LIN {X 0,Y 417.103,Z 397.247,A -85,B 0,C 180,E1 -10165.167,E2 -10165.167} C_VEL
LIN {X 0,Y 417.015,Z 399.098,A -85,B 0,C 180,E1 -10166.135,E2 -10166.135} C_VEL
LIN {X 0,Y 417.032,Z 400.492,A -85,B 0,C 180,E1 -10167.102,E2 -10167.102} C_VEL
LIN {X 0,Y 417.07,Z 401.489,A -85,B 0,C 180,E1 -10168.069,E2 -10168.069} C_VEL
LIN {X 0,Y 417.035,Z 402.093,A -85,B 0,C 180,E1 -10169.035,E2 -10169.035} C_VEL
LIN {X 0,Y 417.032,Z 402.291,A -85,B 0,C 180,E1 -10170,E2 -10170} C_VEL
LIN {X 0,Y 417.071,Z 401.439,A -85,B 0,C 180,E1 -10171.932,E2 -10171.932} C_VEL
LIN {X 0,Y 417.033,Z 400.426,A -85,B 0,C 180,E1 -10172.898,E2 -10172.898} C_VEL
LIN {X 0,Y 417.016,Z 398.993,A -85,B 0,C 180,E1 -10173.866,E2 -10173.866} C_VEL
LIN {X 0,Y 417.09,Z 396.015,A -85,B 0,C 180,E1 -10175.318,E2 -10175.318} C_VEL
LIN {X 0,Y 417.18,Z 391.978,A -85,B 0,C 180,E1 -10176.773,E2 -10176.773} C_VEL
LIN {X 0,Y 417.476,Z 385.766,A -85,B 0,C 180,E1 -10178.471,E2 -10178.471} C_VEL
LIN {X 0,Y 417.86,Z 378.993,A -85,B 0,C 180,E1 -10179.927,E2 -10179.927} C_VEL
LIN {X 0,Y 418.41,Z 370.585,A -85,B 0,C 180,E1 -10181.383,E2 -10181.383} C_VEL
LIN {X 0,Y 419.028,Z 361.919,A -85,B 0,C 180,E1 -10182.594,E2 -10182.594} C_VEL
LIN {X 0,Y 419.708,Z 351.481,A -85,B 0,C 180,E1 -10183.78,E2 -10183.78} C_VEL
LIN {X 0,Y 420.449,Z 340.648,A -85,B 0,C 180,E1 -10184.769,E2 -10184.769} C_VEL
LIN {X 0,Y 421.198,Z 328.876,A -85,B 0,C 180,E1 -10185.609,E2 -10185.609} C_VEL
LIN {X 0,Y 421.835,Z 316.641,A -85,B 0,C 180,E1 -10186.267,E2 -10186.267} C_VEL
LIN {X 0,Y 422.461,Z 303.278,A -85,B 0,C 180,E1 -10186.77,E2 -10186.77} C_VEL
LIN {X 0,Y 422.807,Z 288.187,A -85,B 0,C 180,E1 -10187.098,E2 -10187.098} C_VEL
LIN {X 0,Y 423.445,Z 214.821,A -85,B 0,C 180,E1 -10188.367,E2 -10188.367} C_VEL
LIN {X 0,Y 419.542,Z 189.564,A -85,B 0,C 180,E1 -10188.995,E2 -10188.995} C_VEL
LIN {X 0,Y 420.739,Z 170.933,A -85,B 0,C 180,E1 -10192.594,E2 -10192.594} C_VEL
LIN {X 0,Y 421.255,Z 161.78,A -85,B 0,C 180,E1 -10194.389,E2 -10194.389} C_VEL
LIN {X 0,Y 418.734,Z 148.685,A -85,B 0,C 180,E1 -10197.182,E2 -10197.182} C_VEL
LIN {X 0,Y 418.278,Z 146.385,A -85,B 0,C 180,E1 -10197.686,E2 -10197.686} C_VEL
LIN {X 0,Y 418.243,Z 146.389,A -85,B 0,C 180,E1 -10201.019,E2 -10201.019} C_VEL
LIN {X 0,Y 418.237,Z 146.39,A -85,B 0,C 180,E1 -10203.679,E2 -10203.679} C_VEL
LIN {X 0,Y 418.242,Z 146.387,A -85,B 0,C 180,E1 -10207.224,E2 -10207.224} C_VEL
LIN {X 0,Y 418.211,Z 146.388,A -85,B 0,C 180,E1 -10210.867,E2 -10210.867} C_VEL
LIN {X 0,Y 418.207,Z 146.39,A -85,B 0,C 180,E1 -10213.728,E2 -10213.728} C_VEL
LIN {X 0,Y 418.204,Z 146.388,A -85,B 0,C 180,E1 -10216.447,E2 -10216.447} C_VEL
LIN {X 0,Y 418.215,Z 146.393,A -85,B 0,C 180,E1 -10219.132,E2 -10219.132} C_VEL
LIN {X 0,Y 418.243,Z 146.386,A -85,B 0,C 180,E1 -10222.775,E2 -10222.775} C_VEL
LIN {X 0,Y 418.238,Z 146.384,A -85,B 0,C 180,E1 -10226.321,E2 -10226.321} C_VEL
LIN {X 0,Y 418.244,Z 146.383,A -85,B 0,C 180,E1 -10229.727,E2 -10229.727} C_VEL
LIN {X 0,Y 418.226,Z 146.39,A -85,B 0,C 180,E1 -10233.017,E2 -10233.017} C_VEL
LIN {X 0,Y 418.263,Z 146.382,A -85,B 0,C 180,E1 -10236.217,E2 -10236.217} C_VEL
LIN {X 0,Y 418.252,Z 146.383,A -85,B 0,C 180,E1 -10239.336,E2 -10239.336} C_VEL
LIN {X 0,Y 418.26,Z 146.385,A -85,B 0,C 180,E1 -10242.394,E2 -10242.394} C_VEL
LIN {X 0,Y 418.282,Z 146.378,A -85,B 0,C 180,E1 -10245.402,E2 -10245.402} C_VEL
LIN {X 0,Y 418.318,Z 146.379,A -85,B 0,C 180,E1 -10248.368,E2 -10248.368} C_VEL
LIN {X 0,Y 418.451,Z 146.363,A -85,B 0,C 180,E1 -10252.278,E2 -10252.278} C_VEL
LIN {X 0,Y 418.487,Z 146.358,A -85,B 0,C 180,E1 -10254.216,E2 -10254.216} C_VEL
LIN {X 0,Y 418.538,Z 146.351,A -85,B 0,C 180,E1 -10258.075,E2 -10258.075} C_VEL
LIN {X 0,Y 418.546,Z 146.35,A -85,B 0,C 180,E1 -10259.999,E2 -10259.999} C_VEL
LIN {X 0,Y 418.472,Z 146.355,A -85,B 0,C 180,E1 -10262.887,E2 -10262.887} C_VEL
LIN {X 0,Y 418.44,Z 146.358,A -85,B 0,C 180,E1 -10266.494,E2 -10266.494} C_VEL
LIN {X 0,Y 418.37,Z 146.368,A -85,B 0,C 180,E1 -10268.695,E2 -10268.695} C_VEL
LIN {X 0,Y 418.356,Z 146.369,A -85,B 0,C 180,E1 -10272.613,E2 -10272.613} C_VEL
LIN {X 0,Y 418.249,Z 146.386,A -85,B 0,C 180,E1 -10275.595,E2 -10275.595} C_VEL
LIN {X 0,Y 418.238,Z 146.384,A -85,B 0,C 180,E1 -10278.618,E2 -10278.618} C_VEL
LIN {X 0,Y 418.228,Z 146.392,A -85,B 0,C 180,E1 -10281.696,E2 -10281.696} C_VEL
LIN {X 0,Y 418.244,Z 146.383,A -85,B 0,C 180,E1 -10284.851,E2 -10284.851} C_VEL
LIN {X 0,Y 418.206,Z 146.389,A -85,B 0,C 180,E1 -10288.068,E2 -10288.068} C_VEL
LIN {X 0,Y 418.237,Z 146.386,A -85,B 0,C 180,E1 -10291.018,E2 -10291.018} C_VEL
LIN {X 0,Y 418.231,Z 146.388,A -85,B 0,C 180,E1 -10293.678,E2 -10293.678} C_VEL
LIN {X 0,Y 418.234,Z 146.39,A -85,B 0,C 180,E1 -10297.224,E2 -10297.224} C_VEL
LIN {X 0,Y 418.204,Z 146.391,A -85,B 0,C 180,E1 -10300.866,E2 -10300.866} C_VEL
LIN {X 0,Y 418.199,Z 146.39,A -85,B 0,C 180,E1 -10303.727,E2 -10303.727} C_VEL
LIN {X 0,Y 418.196,Z 146.39,A -85,B 0,C 180,E1 -10306.446,E2 -10306.446} C_VEL
LIN {X 0,Y 418.206,Z 146.394,A -85,B 0,C 180,E1 -10309.131,E2 -10309.131} C_VEL
LIN {X 0,Y 418.233,Z 146.389,A -85,B 0,C 180,E1 -10312.775,E2 -10312.775} C_VEL
LIN {X 0,Y 418.227,Z 146.386,A -85,B 0,C 180,E1 -10316.32,E2 -10316.32} C_VEL
LIN {X 0,Y 418.232,Z 146.384,A -85,B 0,C 180,E1 -10319.727,E2 -10319.727} C_VEL
LIN {X 0,Y 418.204,Z 146.391,A -85,B 0,C 180,E1 -10323.016,E2 -10323.016} C_VEL
LIN {X 0,Y 418.249,Z 146.385,A -85,B 0,C 180,E1 -10326.216,E2 -10326.216} C_VEL
LIN {X 0,Y 418.24,Z 146.384,A -85,B 0,C 180,E1 -10329.336,E2 -10329.336} C_VEL
LIN {X 0,Y 418.24,Z 146.389,A -85,B 0,C 180,E1 -10332.394,E2 -10332.394} C_VEL
LIN {X 0,Y 418.27,Z 146.379,A -85,B 0,C 180,E1 -10335.402,E2 -10335.402} C_VEL
LIN {X 0,Y 418.295,Z 146.383,A -85,B 0,C 180,E1 -10338.368,E2 -10338.368} C_VEL
LIN {X 0,Y 418.439,Z 146.365,A -85,B 0,C 180,E1 -10342.278,E2 -10342.278} C_VEL
LIN {X 0,Y 418.474,Z 146.361,A -85,B 0,C 180,E1 -10344.216,E2 -10344.216} C_VEL
LIN {X 0,Y 418.525,Z 146.354,A -85,B 0,C 180,E1 -10348.075,E2 -10348.075} C_VEL
LIN {X 0,Y 418.493,Z 146.476,A -85,B 0,C 180,E1 -10349.669,E2 -10349.669} C_VEL
LIN {X 0,Y 420.011,Z 155.862,A -85,B 0,C 180,E1 -10351.918,E2 -10351.918} C_VEL
LIN {X 0,Y 419.899,Z 161.158,A -85,B 0,C 180,E1 -10353.094,E2 -10353.094} C_VEL
LIN {X 0,Y 423.923,Z 181.485,A -85,B 0,C 180,E1 -10353.638,E2 -10353.638} C_VEL
LIN {X 0,Y 423.439,Z 219.858,A -85,B 0,C 180,E1 -10354.296,E2 -10354.296} C_VEL
LIN {X 0,Y 422.656,Z 225.699,A -85,B 0,C 180,E1 -10354.367,E2 -10354.367} C_VEL
LIN {X 0,Y 416.911,Z 244.671,A -85,B 0,C 180,E1 -10354.463,E2 -10354.463} C_VEL
LIN {X 0,Y 416.241,Z 250.508,A -85,B 0,C 180,E1 -10354.539,E2 -10354.539} C_VEL
LIN {X 0,Y 415.884,Z 270.871,A -85,B 0,C 180,E1 -10354.938,E2 -10354.938} C_VEL
LIN {X 0,Y 415.455,Z 284.125,A -85,B 0,C 180,E1 -10355.399,E2 -10355.399} C_VEL
LIN {X 0,Y 414.959,Z 297.067,A -85,B 0,C 180,E1 -10356.076,E2 -10356.076} C_VEL
LIN {X 0,Y 414.323,Z 309.401,A -85,B 0,C 180,E1 -10356.942,E2 -10356.942} C_VEL
LIN {X 0,Y 413.565,Z 320.433,A -85,B 0,C 180,E1 -10357.936,E2 -10357.936} C_VEL
LIN {X 0,Y 412.84,Z 330.897,A -85,B 0,C 180,E1 -10359.125,E2 -10359.125} C_VEL
LIN {X 0,Y 412.156,Z 339.445,A -85,B 0,C 180,E1 -10360.314,E2 -10360.314} C_VEL
LIN {X 0,Y 411.556,Z 346.918,A -85,B 0,C 180,E1 -10361.575,E2 -10361.575} C_VEL
LIN {X 0,Y 411.04,Z 353.603,A -85,B 0,C 180,E1 -10362.949,E2 -10362.949} C_VEL
LIN {X 0,Y 410.65,Z 359.189,A -85,B 0,C 180,E1 -10364.368,E2 -10364.368} C_VEL
LIN {X 0,Y 410.33,Z 363.961,A -85,B 0,C 180,E1 -10365.905,E2 -10365.905} C_VEL
LIN {X 0,Y 410.108,Z 367.568,A -85,B 0,C 180,E1 -10367.451,E2 -10367.451} C_VEL
LIN {X 0,Y 409.923,Z 370.608,A -85,B 0,C 180,E1 -10369.449,E2 -10369.449} C_VEL
LIN {X 0,Y 409.812,Z 371.876,A -85,B 0,C 180,E1 -10371.108,E2 -10371.108} C_VEL
LIN {X 0,Y 409.824,Z 372.104,A -85,B 0,C 180,E1 -10372.178,E2 -10372.178} C_VEL
LIN {X 0,Y 409.826,Z 371.839,A -85,B 0,C 180,E1 -10373.23,E2 -10373.23} C_VEL
LIN {X 0,Y 409.901,Z 370.77,A -85,B 0,C 180,E1 -10374.674,E2 -10374.674} C_VEL
LIN {X 0,Y 410.116,Z 368.221,A -85,B 0,C 180,E1 -10376.459,E2 -10376.459} C_VEL
LIN {X 0,Y 410.379,Z 364.648,A -85,B 0,C 180,E1 -10378.096,E2 -10378.096} C_VEL
LIN {X 0,Y 410.693,Z 359.718,A -85,B 0,C 180,E1 -10379.753,E2 -10379.753} C_VEL
LIN {X 0,Y 411.14,Z 353.809,A -85,B 0,C 180,E1 -10381.276,E2 -10381.276} C_VEL
LIN {X 0,Y 411.748,Z 346.273,A -85,B 0,C 180,E1 -10382.815,E2 -10382.815} C_VEL
LIN {X 0,Y 412.465,Z 337.762,A -85,B 0,C 180,E1 -10384.214,E2 -10384.214} C_VEL
LIN {X 0,Y 413.23,Z 328.242,A -85,B 0,C 180,E1 -10385.477,E2 -10385.477} C_VEL
LIN {X 0,Y 414.047,Z 318.004,A -85,B 0,C 180,E1 -10386.569,E2 -10386.569} C_VEL
LIN {X 0,Y 414.795,Z 306.08,A -85,B 0,C 180,E1 -10387.587,E2 -10387.587} C_VEL
LIN {X 0,Y 415.494,Z 294.213,A -85,B 0,C 180,E1 -10388.357,E2 -10388.357} C_VEL
LIN {X 0,Y 416.003,Z 280.901,A -85,B 0,C 180,E1 -10388.992,E2 -10388.992} C_VEL
LIN {X 0,Y 416.363,Z 268.551,A -85,B 0,C 180,E1 -10389.383,E2 -10389.383} C_VEL
LIN {X 0,Y 417.542,Z 181.285,A -85,B 0,C 180,E1 -10390.936,E2 -10390.936} C_VEL
LIN {X 0,Y 413.371,Z 161.521,A -85,B 0,C 180,E1 -10391.534,E2 -10391.534} C_VEL
LIN {X 0,Y 413.138,Z 156.76,A -85,B 0,C 180,E1 -10392.633,E2 -10392.633} C_VEL
LIN {X 0,Y 411.26,Z 147.259,A -85,B 0,C 180,E1 -10394.982,E2 -10394.982} C_VEL
LIN {X 0,Y 411.217,Z 147.263,A -85,B 0,C 180,E1 -10398.201,E2 -10398.201} C_VEL
LIN {X 0,Y 411.227,Z 147.26,A -85,B 0,C 180,E1 -10400.778,E2 -10400.778} C_VEL
LIN {X 0,Y 411.196,Z 147.264,A -85,B 0,C 180,E1 -10404.472,E2 -10404.472} C_VEL
LIN {X 0,Y 411.204,Z 147.262,A -85,B 0,C 180,E1 -10406.874,E2 -10406.874} C_VEL
LIN {X 0,Y 411.231,Z 147.256,A -85,B 0,C 180,E1 -10410.645,E2 -10410.645} C_VEL
LIN {X 0,Y 411.236,Z 147.263,A -85,B 0,C 180,E1 -10413.62,E2 -10413.62} C_VEL
LIN {X 0,Y 411.202,Z 147.264,A -85,B 0,C 180,E1 -10416.853,E2 -10416.853} C_VEL
LIN {X 0,Y 411.214,Z 147.26,A -85,B 0,C 180,E1 -10420.051,E2 -10420.051} C_VEL
LIN {X 0,Y 411.263,Z 147.255,A -85,B 0,C 180,E1 -10423.132,E2 -10423.132} C_VEL
LIN {X 0,Y 411.306,Z 147.248,A -85,B 0,C 180,E1 -10426.897,E2 -10426.897} C_VEL
LIN {X 0,Y 411.292,Z 147.25,A -85,B 0,C 180,E1 -10430.162,E2 -10430.162} C_VEL
LIN {X 0,Y 411.425,Z 147.234,A -85,B 0,C 180,E1 -10433.133,E2 -10433.133} C_VEL
LIN {X 0,Y 411.305,Z 147.242,A -85,B 0,C 180,E1 -10435.1,E2 -10435.1} C_VEL
LIN {X 0,Y 411.511,Z 147.222,A -85,B 0,C 180,E1 -10438.043,E2 -10438.043} C_VEL
LIN {X 0,Y 411.635,Z 147.205,A -85,B 0,C 180,E1 -10440.001,E2 -10440.001} C_VEL
LIN {X 0,Y 411.433,Z 147.231,A -85,B 0,C 180,E1 -10442.938,E2 -10442.938} C_VEL
LIN {X 0,Y 411.435,Z 147.226,A -85,B 0,C 180,E1 -10445.883,E2 -10445.883} C_VEL
LIN {X 0,Y 411.319,Z 147.245,A -85,B 0,C 180,E1 -10448.847,E2 -10448.847} C_VEL
LIN {X 0,Y 411.285,Z 147.245,A -85,B 0,C 180,E1 -10451.833,E2 -10451.833} C_VEL
LIN {X 0,Y 411.235,Z 147.255,A -85,B 0,C 180,E1 -10454.854,E2 -10454.854} C_VEL
LIN {X 0,Y 411.232,Z 147.26,A -85,B 0,C 180,E1 -10457.917,E2 -10457.917} C_VEL
LIN {X 0,Y 411.195,Z 147.259,A -85,B 0,C 180,E1 -10461.035,E2 -10461.035} C_VEL
LIN {X 0,Y 411.192,Z 147.263,A -85,B 0,C 180,E1 -10464.218,E2 -10464.218} C_VEL
LIN {X 0,Y 411.146,Z 147.27,A -85,B 0,C 180,E1 -10467.487,E2 -10467.487} C_VEL
LIN {X 0,Y 411.194,Z 147.26,A -85,B 0,C 180,E1 -10469.714,E2 -10469.714} C_VEL
LIN {X 0,Y 411.205,Z 147.266,A -85,B 0,C 180,E1 -10473.157,E2 -10473.157} C_VEL
LIN {X 0,Y 411.189,Z 147.264,A -85,B 0,C 180,E1 -10476.552,E2 -10476.552} C_VEL
LIN {X 0,Y 411.165,Z 147.269,A -85,B 0,C 180,E1 -10479.72,E2 -10479.72} C_VEL
LIN {X 0,Y 411.163,Z 147.272,A -85,B 0,C 180,E1 -10483.136,E2 -10483.136} C_VEL
LIN {X 0,Y 411.166,Z 147.27,A -85,B 0,C 180,E1 -10485.882,E2 -10485.882} C_VEL
LIN {X 0,Y 411.16,Z 147.27,A -85,B 0,C 180,E1 -10489.493,E2 -10489.493} C_VEL
LIN {X 0,Y 411.186,Z 147.266,A -85,B 0,C 180,E1 -10492.025,E2 -10492.025} C_VEL
LIN {X 0,Y 411.205,Z 147.263,A -85,B 0,C 180,E1 -10495.124,E2 -10495.124} C_VEL
LIN {X 0,Y 411.167,Z 147.269,A -85,B 0,C 180,E1 -10498.003,E2 -10498.003} C_VEL
LIN {X 0,Y 411.196,Z 147.266,A -85,B 0,C 180,E1 -10501.408,E2 -10501.408} C_VEL
LIN {X 0,Y 411.235,Z 147.324,A -85,B 0,C 180,E1 -10501.967,E2 -10501.967} C_VEL
LIN {X 0,Y 413.94,Z 160.534,A -85,B 0,C 180,E1 -10504.884,E2 -10504.884} C_VEL
LIN {X 0,Y 414.362,Z 164.483,A -85,B 0,C 180,E1 -10505.713,E2 -10505.713} C_VEL
LIN {X 0,Y 413.152,Z 181.523,A -85,B 0,C 180,E1 -10509.07,E2 -10509.07} C_VEL
LIN {X 0,Y 412.765,Z 188.745,A -85,B 0,C 180,E1 -10510.484,E2 -10510.484} C_VEL
LIN {X 0,Y 416.97,Z 215.251,A -85,B 0,C 180,E1 -10511.185,E2 -10511.185} C_VEL
LIN {X 0,Y 416.695,Z 257.604,A -85,B 0,C 180,E1 -10511.942,E2 -10511.942} C_VEL
LIN {X 0,Y 416.181,Z 298.233,A -85,B 0,C 180,E1 -10512.685,E2 -10512.685} C_VEL
LIN {X 0,Y 415.509,Z 311.92,A -85,B 0,C 180,E1 -10513.131,E2 -10513.131} C_VEL
LIN {X 0,Y 414.801,Z 324.761,A -85,B 0,C 180,E1 -10513.766,E2 -10513.766} C_VEL
LIN {X 0,Y 413.983,Z 337.3,A -85,B 0,C 180,E1 -10514.618,E2 -10514.618} C_VEL
LIN {X 0,Y 413.137,Z 348.512,A -85,B 0,C 180,E1 -10515.595,E2 -10515.595} C_VEL
LIN {X 0,Y 412.383,Z 358.602,A -85,B 0,C 180,E1 -10516.699,E2 -10516.699} C_VEL
LIN {X 0,Y 411.747,Z 367.741,A -85,B 0,C 180,E1 -10517.931,E2 -10517.931} C_VEL
LIN {X 0,Y 410.957,Z 376.66,A -85,B 0,C 180,E1 -10519.407,E2 -10519.407} C_VEL
LIN {X 0,Y 410.544,Z 383.834,A -85,B 0,C 180,E1 -10520.889,E2 -10520.889} C_VEL
LIN {X 0,Y 410.183,Z 390.377,A -85,B 0,C 180,E1 -10522.617,E2 -10522.617} C_VEL
LIN {X 0,Y 409.998,Z 394.707,A -85,B 0,C 180,E1 -10524.097,E2 -10524.097} C_VEL
LIN {X 0,Y 410.01,Z 397.008,A -85,B 0,C 180,E1 -10525.084,E2 -10525.084} C_VEL
LIN {X 0,Y 409.933,Z 398.853,A -85,B 0,C 180,E1 -10526.068,E2 -10526.068} C_VEL
LIN {X 0,Y 409.998,Z 401.238,A -85,B 0,C 180,E1 -10528.036,E2 -10528.036} C_VEL
LIN {X 0,Y 409.958,Z 401.839,A -85,B 0,C 180,E1 -10529.018,E2 -10529.018} C_VEL
LIN {X 0,Y 409.953,Z 402.031,A -85,B 0,C 180,E1 -10530,E2 -10530} C_VEL
LIN {X 0,Y 409.998,Z 401.172,A -85,B 0,C 180,E1 -10531.965,E2 -10531.965} C_VEL
LIN {X 0,Y 409.932,Z 400.153,A -85,B 0,C 180,E1 -10532.948,E2 -10532.948} C_VEL
LIN {X 0,Y 409.933,Z 398.713,A -85,B 0,C 180,E1 -10533.932,E2 -10533.932} C_VEL
LIN {X 0,Y 409.988,Z 395.726,A -85,B 0,C 180,E1 -10535.41,E2 -10535.41} C_VEL
LIN {X 0,Y 410.099,Z 391.681,A -85,B 0,C 180,E1 -10536.89,E2 -10536.89} C_VEL
LIN {X 0,Y 410.409,Z 385.455,A -85,B 0,C 180,E1 -10538.618,E2 -10538.618} C_VEL
LIN {X 0,Y 410.831,Z 378.671,A -85,B 0,C 180,E1 -10540.099,E2 -10540.099} C_VEL
LIN {X 0,Y 411.429,Z 370.245,A -85,B 0,C 180,E1 -10541.579,E2 -10541.579} C_VEL
LIN {X 0,Y 412.028,Z 361.556,A -85,B 0,C 180,E1 -10542.812,E2 -10542.812} C_VEL
LIN {X 0,Y 412.799,Z 351.098,A -85,B 0,C 180,E1 -10544.016,E2 -10544.016} C_VEL
LIN {X 0,Y 413.558,Z 340.238,A -85,B 0,C 180,E1 -10545.02,E2 -10545.02} C_VEL
LIN {X 0,Y 414.357,Z 328.406,A -85,B 0,C 180,E1 -10545.873,E2 -10545.873} C_VEL
LIN {X 0,Y 415.015,Z 316.106,A -85,B 0,C 180,E1 -10546.542,E2 -10546.542} C_VEL
LIN {X 0,Y 415.686,Z 302.595,A -85,B 0,C 180,E1 -10547.052,E2 -10547.052} C_VEL
LIN {X 0,Y 416.012,Z 287.175,A -85,B 0,C 180,E1 -10547.386,E2 -10547.386} C_VEL
LIN {X 0,Y 416.647,Z 215.378,A -85,B 0,C 180,E1 -10548.65,E2 -10548.65} C_VEL
LIN {X 0,Y 412.633,Z 189.318,A -85,B 0,C 180,E1 -10549.311,E2 -10549.311} C_VEL
LIN {X 0,Y 413.857,Z 170.608,A -85,B 0,C 180,E1 -10552.991,E2 -10552.991} C_VEL
LIN {X 0,Y 414.29,Z 162.755,A -85,B 0,C 180,E1 -10554.559,E2 -10554.559} C_VEL
LIN {X 0,Y 411.687,Z 149.488,A -85,B 0,C 180,E1 -10557.447,E2 -10557.447} C_VEL
LIN {X 0,Y 411.224,Z 147.263,A -85,B 0,C 180,E1 -10557.965,E2 -10557.965} C_VEL
LIN {X 0,Y 411.186,Z 147.268,A -85,B 0,C 180,E1 -10561.283,E2 -10561.283} C_VEL
LIN {X 0,Y 411.197,Z 147.261,A -85,B 0,C 180,E1 -10564.335,E2 -10564.335} C_VEL
LIN {X 0,Y 411.193,Z 147.261,A -85,B 0,C 180,E1 -10566.742,E2 -10566.742} C_VEL
LIN {X 0,Y 411.174,Z 147.267,A -85,B 0,C 180,E1 -10569.72,E2 -10569.72} C_VEL
LIN {X 0,Y 411.167,Z 147.269,A -85,B 0,C 180,E1 -10573.135,E2 -10573.135} C_VEL
LIN {X 0,Y 411.168,Z 147.265,A -85,B 0,C 180,E1 -10575.882,E2 -10575.882} C_VEL
LIN {X 0,Y 411.168,Z 147.268,A -85,B 0,C 180,E1 -10579.493,E2 -10579.493} C_VEL
LIN {X 0,Y 411.192,Z 147.261,A -85,B 0,C 180,E1 -10582.025,E2 -10582.025} C_VEL
LIN {X 0,Y 411.198,Z 147.262,A -85,B 0,C 180,E1 -10585.665,E2 -10585.665} C_VEL
LIN {X 0,Y 411.192,Z 147.266,A -85,B 0,C 180,E1 -10589.152,E2 -10589.152} C_VEL
LIN {X 0,Y 411.183,Z 147.264,A -85,B 0,C 180,E1 -10591.407,E2 -10591.407} C_VEL
LIN {X 0,Y 411.217,Z 147.264,A -85,B 0,C 180,E1 -10594.934,E2 -10594.934} C_VEL
LIN {X 0,Y 411.207,Z 147.259,A -85,B 0,C 180,E1 -10597.913,E2 -10597.913} C_VEL
LIN {X 0,Y 411.22,Z 147.261,A -85,B 0,C 180,E1 -10601.051,E2 -10601.051} C_VEL
LIN {X 0,Y 411.215,Z 147.26,A -85,B 0,C 180,E1 -10604.129,E2 -10604.129} C_VEL
LIN {X 0,Y 411.309,Z 147.248,A -85,B 0,C 180,E1 -10607.165,E2 -10607.165} C_VEL
LIN {X 0,Y 411.29,Z 147.253,A -85,B 0,C 180,E1 -10610.16,E2 -10610.16} C_VEL
LIN {X 0,Y 411.395,Z 147.236,A -85,B 0,C 180,E1 -10613.131,E2 -10613.131} C_VEL
LIN {X 0,Y 411.293,Z 147.249,A -85,B 0,C 180,E1 -10615.098,E2 -10615.098} C_VEL
LIN {X 0,Y 411.507,Z 147.226,A -85,B 0,C 180,E1 -10618.042,E2 -10618.042} C_VEL
LIN {X 0,Y 411.384,Z 147.238,A -85,B 0,C 180,E1 -10620.978,E2 -10620.978} C_VEL
LIN {X 0,Y 411.431,Z 147.232,A -85,B 0,C 180,E1 -10622.937,E2 -10622.937} C_VEL
LIN {X 0,Y 411.393,Z 147.236,A -85,B 0,C 180,E1 -10626.867,E2 -10626.867} C_VEL
LIN {X 0,Y 411.279,Z 147.256,A -85,B 0,C 180,E1 -10629.838,E2 -10629.838} C_VEL
LIN {X 0,Y 411.307,Z 147.247,A -85,B 0,C 180,E1 -10633.102,E2 -10633.102} C_VEL
LIN {X 0,Y 411.209,Z 147.259,A -85,B 0,C 180,E1 -10636.89,E2 -10636.89} C_VEL
LIN {X 0,Y 411.205,Z 147.264,A -85,B 0,C 180,E1 -10639.987,E2 -10639.987} C_VEL
LIN {X 0,Y 411.187,Z 147.263,A -85,B 0,C 180,E1 -10643.147,E2 -10643.147} C_VEL
LIN {X 0,Y 411.171,Z 147.264,A -85,B 0,C 180,E1 -10646.384,E2 -10646.384} C_VEL
LIN {X 0,Y 411.194,Z 147.266,A -85,B 0,C 180,E1 -10649.712,E2 -10649.712} C_VEL
LIN {X 0,Y 411.203,Z 147.264,A -85,B 0,C 180,E1 -10653.155,E2 -10653.155} C_VEL
LIN {X 0,Y 411.189,Z 147.262,A -85,B 0,C 180,E1 -10656.551,E2 -10656.551} C_VEL
LIN {X 0,Y 411.165,Z 147.267,A -85,B 0,C 180,E1 -10659.719,E2 -10659.719} C_VEL
LIN {X 0,Y 411.159,Z 147.272,A -85,B 0,C 180,E1 -10663.134,E2 -10663.134} C_VEL
LIN {X 0,Y 411.16,Z 147.266,A -85,B 0,C 180,E1 -10665.881,E2 -10665.881} C_VEL
LIN {X 0,Y 411.159,Z 147.267,A -85,B 0,C 180,E1 -10669.493,E2 -10669.493} C_VEL
LIN {X 0,Y 411.182,Z 147.262,A -85,B 0,C 180,E1 -10672.024,E2 -10672.024} C_VEL
LIN {X 0,Y 411.187,Z 147.262,A -85,B 0,C 180,E1 -10675.664,E2 -10675.664} C_VEL
LIN {X 0,Y 411.181,Z 147.266,A -85,B 0,C 180,E1 -10679.151,E2 -10679.151} C_VEL
LIN {X 0,Y 411.165,Z 147.265,A -85,B 0,C 180,E1 -10681.406,E2 -10681.406} C_VEL
LIN {X 0,Y 411.181,Z 147.266,A -85,B 0,C 180,E1 -10684.94,E2 -10684.94} C_VEL
LIN {X 0,Y 411.195,Z 147.262,A -85,B 0,C 180,E1 -10687.913,E2 -10687.913} C_VEL
LIN {X 0,Y 411.204,Z 147.261,A -85,B 0,C 180,E1 -10691.05,E2 -10691.05} C_VEL
LIN {X 0,Y 411.202,Z 147.263,A -85,B 0,C 180,E1 -10694.129,E2 -10694.129} C_VEL
LIN {X 0,Y 411.295,Z 147.249,A -85,B 0,C 180,E1 -10697.165,E2 -10697.165} C_VEL
LIN {X 0,Y 411.268,Z 147.257,A -85,B 0,C 180,E1 -10700.16,E2 -10700.16} C_VEL
LIN {X 0,Y 411.382,Z 147.238,A -85,B 0,C 180,E1 -10703.131,E2 -10703.131} C_VEL
LIN {X 0,Y 411.28,Z 147.25,A -85,B 0,C 180,E1 -10705.098,E2 -10705.098} C_VEL
LIN {X 0,Y 411.494,Z 147.23,A -85,B 0,C 180,E1 -10708.042,E2 -10708.042} C_VEL
LIN {X 0,Y 411.432,Z 147.383,A -85,B 0,C 180,E1 -10709.449,E2 -10709.449} C_VEL
LIN {X 0,Y 413.085,Z 157.68,A -85,B 0,C 180,E1 -10711.95,E2 -10711.95} C_VEL
LIN {X 0,Y 412.963,Z 161.276,A -85,B 0,C 180,E1 -10712.774,E2 -10712.774} C_VEL
LIN {X 0,Y 417.126,Z 181.324,A -85,B 0,C 180,E1 -10713.332,E2 -10713.332} C_VEL
LIN {X 0,Y 416.241,Z 250.508,A -85,B 0,C 180,E1 -10714.539,E2 -10714.539} C_VEL
LIN {X 0,Y 415.555,Z 256.355,A -85,B 0,C 180,E1 -10714.613,E2 -10714.613} C_VEL
LIN {X 0,Y 412.642,Z 265.838,A -85,B 0,C 180,E1 -10714.675,E2 -10714.675} C_VEL
LIN {X 0,Y 409.627,Z 275.225,A -85,B 0,C 180,E1 -10714.807,E2 -10714.807} C_VEL
LIN {X 0,Y 408.774,Z 280.917,A -85,B 0,C 180,E1 -10714.987,E2 -10714.987} C_VEL
LIN {X 0,Y 408.273,Z 294.011,A -85,B 0,C 180,E1 -10715.618,E2 -10715.618} C_VEL
LIN {X 0,Y 407.632,Z 306.348,A -85,B 0,C 180,E1 -10716.434,E2 -10716.434} C_VEL
LIN {X 0,Y 406.865,Z 318.034,A -85,B 0,C 180,E1 -10717.444,E2 -10717.444} C_VEL
LIN {X 0,Y 406.124,Z 328.54,A -85,B 0,C 180,E1 -10718.584,E2 -10718.584} C_VEL
LIN {X 0,Y 405.389,Z 337.175,A -85,B 0,C 180,E1 -10719.735,E2 -10719.735} C_VEL
LIN {X 0,Y 404.614,Z 346.437,A -85,B 0,C 180,E1 -10721.268,E2 -10721.268} C_VEL
LIN {X 0,Y 404.006,Z 354.19,A -85,B 0,C 180,E1 -10722.878,E2 -10722.878} C_VEL
LIN {X 0,Y 403.501,Z 360.707,A -85,B 0,C 180,E1 -10724.629,E2 -10724.629} C_VEL
LIN {X 0,Y 403.217,Z 365.175,A -85,B 0,C 180,E1 -10726.193,E2 -10726.193} C_VEL
LIN {X 0,Y 403.05,Z 367.544,A -85,B 0,C 180,E1 -10727.243,E2 -10727.243} C_VEL
LIN {X 0,Y 402.891,Z 369.409,A -85,B 0,C 180,E1 -10728.3,E2 -10728.3} C_VEL
LIN {X 0,Y 402.824,Z 371.065,A -85,B 0,C 180,E1 -10729.591,E2 -10729.591} C_VEL
LIN {X 0,Y 402.711,Z 372.269,A -85,B 0,C 180,E1 -10731.499,E2 -10731.499} C_VEL
LIN {X 0,Y 402.731,Z 372.307,A -85,B 0,C 180,E1 -10732.577,E2 -10732.577} C_VEL
LIN {X 0,Y 402.738,Z 371.912,A -85,B 0,C 180,E1 -10733.663,E2 -10733.663} C_VEL
LIN {X 0,Y 402.827,Z 370.869,A -85,B 0,C 180,E1 -10734.878,E2 -10734.878} C_VEL
LIN {X 0,Y 402.953,Z 369.621,A -85,B 0,C 180,E1 -10735.851,E2 -10735.851} C_VEL
LIN {X 0,Y 403.162,Z 367.125,A -85,B 0,C 180,E1 -10737.249,E2 -10737.249} C_VEL
LIN {X 0,Y 403.474,Z 362.237,A -85,B 0,C 180,E1 -10739.191,E2 -10739.191} C_VEL
LIN {X 0,Y 403.952,Z 356.386,A -85,B 0,C 180,E1 -10740.88,E2 -10740.88} C_VEL
LIN {X 0,Y 404.578,Z 348.813,A -85,B 0,C 180,E1 -10742.582,E2 -10742.582} C_VEL
LIN {X 0,Y 405.313,Z 340.854,A -85,B 0,C 180,E1 -10744.001,E2 -10744.001} C_VEL
LIN {X 0,Y 406.086,Z 331.567,A -85,B 0,C 180,E1 -10745.337,E2 -10745.337} C_VEL
LIN {X 0,Y 406.962,Z 320.941,A -85,B 0,C 180,E1 -10746.569,E2 -10746.569} C_VEL
LIN {X 0,Y 407.756,Z 310.342,A -85,B 0,C 180,E1 -10747.549,E2 -10747.549} C_VEL
LIN {X 0,Y 408.509,Z 299.389,A -85,B 0,C 180,E1 -10748.347,E2 -10748.347} C_VEL
LIN {X 0,Y 409.056,Z 286.292,A -85,B 0,C 180,E1 -10749.074,E2 -10749.074} C_VEL
LIN {X 0,Y 409.469,Z 274.185,A -85,B 0,C 180,E1 -10749.544,E2 -10749.544} C_VEL
LIN {X 0,Y 409.802,Z 259.096,A -85,B 0,C 180,E1 -10749.884,E2 -10749.884} C_VEL
LIN {X 0,Y 410.832,Z 182.187,A -85,B 0,C 180,E1 -10751.26,E2 -10751.26} C_VEL
LIN {X 0,Y 406.469,Z 161.878,A -85,B 0,C 180,E1 -10751.875,E2 -10751.875} C_VEL
LIN {X 0,Y 406.124,Z 157.65,A -85,B 0,C 180,E1 -10752.878,E2 -10752.878} C_VEL
LIN {X 0,Y 404.181,Z 148.139,A -85,B 0,C 180,E1 -10755.266,E2 -10755.266} C_VEL
LIN {X 0,Y 404.188,Z 148.138,A -85,B 0,C 180,E1 -10758.39,E2 -10758.39} C_VEL
LIN {X 0,Y 404.158,Z 148.144,A -85,B 0,C 180,E1 -10761.492,E2 -10761.492} C_VEL
LIN {X 0,Y 404.182,Z 148.139,A -85,B 0,C 180,E1 -10764.985,E2 -10764.985} C_VEL
LIN {X 0,Y 404.139,Z 148.141,A -85,B 0,C 180,E1 -10768.555,E2 -10768.555} C_VEL
LIN {X 0,Y 404.194,Z 148.136,A -85,B 0,C 180,E1 -10772.001,E2 -10772.001} C_VEL
LIN {X 0,Y 404.176,Z 148.14,A -85,B 0,C 180,E1 -10775.335,E2 -10775.335} C_VEL
LIN {X 0,Y 404.138,Z 148.144,A -85,B 0,C 180,E1 -10778.582,E2 -10778.582} C_VEL
LIN {X 0,Y 404.204,Z 148.133,A -85,B 0,C 180,E1 -10781.763,E2 -10781.763} C_VEL
LIN {X 0,Y 404.206,Z 148.139,A -85,B 0,C 180,E1 -10784.883,E2 -10784.883} C_VEL
LIN {X 0,Y 404.257,Z 148.125,A -85,B 0,C 180,E1 -10787.959,E2 -10787.959} C_VEL
LIN {X 0,Y 404.267,Z 148.122,A -85,B 0,C 180,E1 -10790.999,E2 -10790.999} C_VEL
LIN {X 0,Y 404.394,Z 148.109,A -85,B 0,C 180,E1 -10794.015,E2 -10794.015} C_VEL
LIN {X 0,Y 404.48,Z 148.097,A -85,B 0,C 180,E1 -10798.009,E2 -10798.009} C_VEL
LIN {X 0,Y 404.605,Z 148.081,A -85,B 0,C 180,E1 -10800.001,E2 -10800.001} C_VEL
LIN {X 0,Y 404.393,Z 148.107,A -85,B 0,C 180,E1 -10802.989,E2 -10802.989} C_VEL
LIN {X 0,Y 404.383,Z 148.104,A -85,B 0,C 180,E1 -10805.986,E2 -10805.986} C_VEL
LIN {X 0,Y 404.266,Z 148.123,A -85,B 0,C 180,E1 -10809.002,E2 -10809.002} C_VEL
LIN {X 0,Y 404.258,Z 148.123,A -85,B 0,C 180,E1 -10812.042,E2 -10812.042} C_VEL
LIN {X 0,Y 404.179,Z 148.134,A -85,B 0,C 180,E1 -10815.12,E2 -10815.12} C_VEL
LIN {X 0,Y 404.196,Z 148.136,A -85,B 0,C 180,E1 -10818.239,E2 -10818.239} C_VEL
LIN {X 0,Y 404.137,Z 148.138,A -85,B 0,C 180,E1 -10821.42,E2 -10821.42} C_VEL
LIN {X 0,Y 404.137,Z 148.141,A -85,B 0,C 180,E1 -10824.669,E2 -10824.669} C_VEL
LIN {X 0,Y 404.103,Z 148.147,A -85,B 0,C 180,E1 -10828.007,E2 -10828.007} C_VEL
LIN {X 0,Y 404.141,Z 148.135,A -85,B 0,C 180,E1 -10830.286,E2 -10830.286} C_VEL
LIN {X 0,Y 404.138,Z 148.139,A -85,B 0,C 180,E1 -10833.814,E2 -10833.814} C_VEL
LIN {X 0,Y 404.132,Z 148.146,A -85,B 0,C 180,E1 -10836.874,E2 -10836.874} C_VEL
LIN {X 0,Y 404.119,Z 148.145,A -85,B 0,C 180,E1 -10840.075,E2 -10840.075} C_VEL
LIN {X 0,Y 404.143,Z 148.147,A -85,B 0,C 180,E1 -10843.082,E2 -10843.082} C_VEL
LIN {X 0,Y 404.123,Z 148.148,A -85,B 0,C 180,E1 -10845.922,E2 -10845.922} C_VEL
LIN {X 0,Y 404.104,Z 148.152,A -85,B 0,C 180,E1 -10848.633,E2 -10848.633} C_VEL
LIN {X 0,Y 404.141,Z 148.143,A -85,B 0,C 180,E1 -10851.495,E2 -10851.495} C_VEL
LIN {X 0,Y 404.18,Z 148.139,A -85,B 0,C 180,E1 -10854.983,E2 -10854.983} C_VEL
LIN {X 0,Y 404.141,Z 148.143,A -85,B 0,C 180,E1 -10858.443,E2 -10858.443} C_VEL
LIN {X 0,Y 404.212,Z 148.305,A -85,B 0,C 180,E1 -10861.684,E2 -10861.684} C_VEL
LIN {X 0,Y 406.972,Z 161.671,A -85,B 0,C 180,E1 -10864.697,E2 -10864.697} C_VEL
LIN {X 0,Y 407.45,Z 165.622,A -85,B 0,C 180,E1 -10865.546,E2 -10865.546} C_VEL
LIN {X 0,Y 406.28,Z 181.332,A -85,B 0,C 180,E1 -10868.699,E2 -10868.699} C_VEL
LIN {X 0,Y 405.869,Z 188.476,A -85,B 0,C 180,E1 -10870.122,E2 -10870.122} C_VEL
LIN {X 0,Y 409.976,Z 213.769,A -85,B 0,C 180,E1 -10870.813,E2 -10870.813} C_VEL
LIN {X 0,Y 410.429,Z 220.076,A -85,B 0,C 180,E1 -10870.953,E2 -10870.953} C_VEL
LIN {X 0,Y 409.467,Z 297.344,A -85,B 0,C 180,E1 -10872.359,E2 -10872.359} C_VEL
LIN {X 0,Y 408.792,Z 310.473,A -85,B 0,C 180,E1 -10872.781,E2 -10872.781} C_VEL
LIN {X 0,Y 408.063,Z 323.697,A -85,B 0,C 180,E1 -10873.426,E2 -10873.426} C_VEL
LIN {X 0,Y 407.266,Z 335.624,A -85,B 0,C 180,E1 -10874.229,E2 -10874.229} C_VEL
LIN {X 0,Y 406.331,Z 347.34,A -85,B 0,C 180,E1 -10875.245,E2 -10875.245} C_VEL
LIN {X 0,Y 405.575,Z 357.445,A -85,B 0,C 180,E1 -10876.346,E2 -10876.346} C_VEL
LIN {X 0,Y 404.913,Z 365.897,A -85,B 0,C 180,E1 -10877.47,E2 -10877.47} C_VEL
LIN {X 0,Y 404.055,Z 375.086,A -85,B 0,C 180,E1 -10878.97,E2 -10878.97} C_VEL
LIN {X 0,Y 403.567,Z 382.503,A -85,B 0,C 180,E1 -10880.477,E2 -10880.477} C_VEL
LIN {X 0,Y 403.206,Z 388.464,A -85,B 0,C 180,E1 -10881.985,E2 -10881.985} C_VEL
LIN {X 0,Y 402.965,Z 393.173,A -85,B 0,C 180,E1 -10883.491,E2 -10883.491} C_VEL
LIN {X 0,Y 402.919,Z 396.768,A -85,B 0,C 180,E1 -10884.997,E2 -10884.997} C_VEL
LIN {X 0,Y 402.853,Z 398.608,A -85,B 0,C 180,E1 -10885.999,E2 -10885.999} C_VEL
LIN {X 0,Y 402.908,Z 400.987,A -85,B 0,C 180,E1 -10888.001,E2 -10888.001} C_VEL
LIN {X 0,Y 402.885,Z 401.586,A -85,B 0,C 180,E1 -10889.001,E2 -10889.001} C_VEL
LIN {X 0,Y 402.876,Z 401.77,A -85,B 0,C 180,E1 -10890,E2 -10890} C_VEL
LIN {X 0,Y 402.885,Z 401.531,A -85,B 0,C 180,E1 -10891,E2 -10891} C_VEL
LIN {X 0,Y 402.908,Z 400.904,A -85,B 0,C 180,E1 -10891.999,E2 -10891.999} C_VEL
LIN {X 0,Y 402.832,Z 399.881,A -85,B 0,C 180,E1 -10893,E2 -10893} C_VEL
LIN {X 0,Y 402.853,Z 398.433,A -85,B 0,C 180,E1 -10894.002,E2 -10894.002} C_VEL
LIN {X 0,Y 402.887,Z 395.438,A -85,B 0,C 180,E1 -10895.506,E2 -10895.506} C_VEL
LIN {X 0,Y 403.043,Z 391.385,A -85,B 0,C 180,E1 -10897.011,E2 -10897.011} C_VEL
LIN {X 0,Y 403.365,Z 385.146,A -85,B 0,C 180,E1 -10898.769,E2 -10898.769} C_VEL
LIN {X 0,Y 403.784,Z 378.348,A -85,B 0,C 180,E1 -10900.277,E2 -10900.277} C_VEL
LIN {X 0,Y 404.436,Z 369.903,A -85,B 0,C 180,E1 -10901.782,E2 -10901.782} C_VEL
LIN {X 0,Y 405.062,Z 361.194,A -85,B 0,C 180,E1 -10903.036,E2 -10903.036} C_VEL
LIN {X 0,Y 405.897,Z 350.477,A -85,B 0,C 180,E1 -10904.285,E2 -10904.285} C_VEL
LIN {X 0,Y 406.681,Z 339.827,A -85,B 0,C 180,E1 -10905.281,E2 -10905.281} C_VEL
LIN {X 0,Y 407.508,Z 327.935,A -85,B 0,C 180,E1 -10906.147,E2 -10906.147} C_VEL
LIN {X 0,Y 408.197,Z 315.57,A -85,B 0,C 180,E1 -10906.826,E2 -10906.826} C_VEL
LIN {X 0,Y 408.857,Z 302.905,A -85,B 0,C 180,E1 -10907.313,E2 -10907.313} C_VEL
LIN {X 0,Y 409.223,Z 287.943,A -85,B 0,C 180,E1 -10907.652,E2 -10907.652} C_VEL
LIN {X 0,Y 409.875,Z 216.127,A -85,B 0,C 180,E1 -10908.938,E2 -10908.938} C_VEL
LIN {X 0,Y 405.72,Z 188.991,A -85,B 0,C 180,E1 -10909.653,E2 -10909.653} C_VEL
LIN {X 0,Y 406.903,Z 171.583,A -85,B 0,C 180,E1 -10913.138,E2 -10913.138} C_VEL
LIN {X 0,Y 407.292,Z 163.732,A -85,B 0,C 180,E1 -10914.737,E2 -10914.737} C_VEL
LIN {X 0,Y 404.684,Z 150.546,A -85,B 0,C 180,E1 -10917.661,E2 -10917.661} C_VEL
LIN {X 0,Y 404.187,Z 148.138,A -85,B 0,C 180,E1 -10918.212,E2 -10918.212} C_VEL
LIN {X 0,Y 404.143,Z 148.146,A -85,B 0,C 180,E1 -10921.558,E2 -10921.558} C_VEL
LIN {X 0,Y 404.182,Z 148.136,A -85,B 0,C 180,E1 -10925.017,E2 -10925.017} C_VEL
LIN {X 0,Y 404.139,Z 148.14,A -85,B 0,C 180,E1 -10928.759,E2 -10928.759} C_VEL
LIN {X 0,Y 404.111,Z 148.148,A -85,B 0,C 180,E1 -10931.597,E2 -10931.597} C_VEL
LIN {X 0,Y 404.148,Z 148.139,A -85,B 0,C 180,E1 -10934.522,E2 -10934.522} C_VEL
LIN {X 0,Y 404.126,Z 148.148,A -85,B 0,C 180,E1 -10937.293,E2 -10937.293} C_VEL
LIN {X 0,Y 404.137,Z 148.14,A -85,B 0,C 180,E1 -10939.951,E2 -10939.951} C_VEL
LIN {X 0,Y 404.14,Z 148.147,A -85,B 0,C 180,E1 -10943.125,E2 -10943.125} C_VEL
LIN {X 0,Y 404.143,Z 148.139,A -85,B 0,C 180,E1 -10946.187,E2 -10946.187} C_VEL
LIN {X 0,Y 404.147,Z 148.139,A -85,B 0,C 180,E1 -10949.714,E2 -10949.714} C_VEL
LIN {X 0,Y 404.13,Z 148.145,A -85,B 0,C 180,E1 -10953.117,E2 -10953.117} C_VEL
LIN {X 0,Y 404.154,Z 148.141,A -85,B 0,C 180,E1 -10956.424,E2 -10956.424} C_VEL
LIN {X 0,Y 404.197,Z 148.133,A -85,B 0,C 180,E1 -10959.874,E2 -10959.874} C_VEL
LIN {X 0,Y 404.179,Z 148.138,A -85,B 0,C 180,E1 -10963.012,E2 -10963.012} C_VEL
LIN {X 0,Y 404.288,Z 148.124,A -85,B 0,C 180,E1 -10966.938,E2 -10966.938} C_VEL
LIN {X 0,Y 404.257,Z 148.127,A -85,B 0,C 180,E1 -10969.987,E2 -10969.987} C_VEL
LIN {X 0,Y 404.345,Z 148.115,A -85,B 0,C 180,E1 -10973.011,E2 -10973.011} C_VEL
LIN {X 0,Y 404.265,Z 148.125,A -85,B 0,C 180,E1 -10975.013,E2 -10975.013} C_VEL
LIN {X 0,Y 404.475,Z 148.102,A -85,B 0,C 180,E1 -10978.008,E2 -10978.008} C_VEL
LIN {X 0,Y 404.354,Z 148.113,A -85,B 0,C 180,E1 -10980.995,E2 -10980.995} C_VEL
LIN {X 0,Y 404.39,Z 148.109,A -85,B 0,C 180,E1 -10982.988,E2 -10982.988} C_VEL
LIN {X 0,Y 404.344,Z 148.114,A -85,B 0,C 180,E1 -10986.988,E2 -10986.988} C_VEL
LIN {X 0,Y 404.246,Z 148.133,A -85,B 0,C 180,E1 -10990.011,E2 -10990.011} C_VEL
LIN {X 0,Y 404.27,Z 148.124,A -85,B 0,C 180,E1 -10993.21,E2 -10993.21} C_VEL
LIN {X 0,Y 404.157,Z 148.138,A -85,B 0,C 180,E1 -10996.977,E2 -10996.977} C_VEL
LIN {X 0,Y 404.152,Z 148.139,A -85,B 0,C 180,E1 -11000.351,E2 -11000.351} C_VEL
LIN {X 0,Y 404.148,Z 148.145,A -85,B 0,C 180,E1 -11003.575,E2 -11003.575} C_VEL
LIN {X 0,Y 404.103,Z 148.145,A -85,B 0,C 180,E1 -11006.883,E2 -11006.883} C_VEL
LIN {X 0,Y 404.141,Z 148.14,A -85,B 0,C 180,E1 -11010.284,E2 -11010.284} C_VEL
LIN {X 0,Y 404.137,Z 148.143,A -85,B 0,C 180,E1 -11013.812,E2 -11013.812} C_VEL
LIN {X 0,Y 404.131,Z 148.143,A -85,B 0,C 180,E1 -11016.873,E2 -11016.873} C_VEL
LIN {X 0,Y 404.114,Z 148.143,A -85,B 0,C 180,E1 -11020.074,E2 -11020.074} C_VEL
LIN {X 0,Y 404.139,Z 148.146,A -85,B 0,C 180,E1 -11023.081,E2 -11023.081} C_VEL
LIN {X 0,Y 404.117,Z 148.143,A -85,B 0,C 180,E1 -11025.921,E2 -11025.921} C_VEL
LIN {X 0,Y 404.099,Z 148.147,A -85,B 0,C 180,E1 -11028.632,E2 -11028.632} C_VEL
LIN {X 0,Y 404.137,Z 148.142,A -85,B 0,C 180,E1 -11031.493,E2 -11031.493} C_VEL
LIN {X 0,Y 404.169,Z 148.142,A -85,B 0,C 180,E1 -11034.982,E2 -11034.982} C_VEL
LIN {X 0,Y 404.132,Z 148.144,A -85,B 0,C 180,E1 -11038.442,E2 -11038.442} C_VEL
LIN {X 0,Y 404.143,Z 148.145,A -85,B 0,C 180,E1 -11040.861,E2 -11040.861} C_VEL
LIN {X 0,Y 404.146,Z 148.145,A -85,B 0,C 180,E1 -11044.722,E2 -11044.722} C_VEL
LIN {X 0,Y 404.159,Z 148.137,A -85,B 0,C 180,E1 -11047.507,E2 -11047.507} C_VEL
LIN {X 0,Y 404.15,Z 148.143,A -85,B 0,C 180,E1 -11050.706,E2 -11050.706} C_VEL
LIN {X 0,Y 404.172,Z 148.137,A -85,B 0,C 180,E1 -11053.846,E2 -11053.846} C_VEL
LIN {X 0,Y 404.276,Z 148.124,A -85,B 0,C 180,E1 -11056.938,E2 -11056.938} C_VEL
LIN {X 0,Y 404.235,Z 148.131,A -85,B 0,C 180,E1 -11059.987,E2 -11059.987} C_VEL
LIN {X 0,Y 404.332,Z 148.116,A -85,B 0,C 180,E1 -11063.011,E2 -11063.011} C_VEL
LIN {X 0,Y 404.252,Z 148.126,A -85,B 0,C 180,E1 -11065.013,E2 -11065.013} C_VEL
LIN {X 0,Y 404.463,Z 148.105,A -85,B 0,C 180,E1 -11068.008,E2 -11068.008} C_VEL
LIN {X 0,Y 404.348,Z 148.2,A -85,B 0,C 180,E1 -11069.191,E2 -11069.191} C_VEL
LIN {X 0,Y 406.005,Z 157.432,A -85,B 0,C 180,E1 -11071.488,E2 -11071.488} C_VEL
LIN {X 0,Y 406.06,Z 161.497,A -85,B 0,C 180,E1 -11072.447,E2 -11072.447} C_VEL
LIN {X 0,Y 410.375,Z 182.359,A -85,B 0,C 180,E1 -11073.042,E2 -11073.042} C_VEL
LIN {X 0,Y 409.161,Z 269.377,A -85,B 0,C 180,E1 -11074.614,E2 -11074.614} C_VEL
LIN {X 0,Y 408.774,Z 280.917,A -85,B 0,C 180,E1 -11074.987,E2 -11074.987} C_VEL
LIN {X 0,Y 407.876,Z 286.68,A -85,B 0,C 180,E1 -11075.207,E2 -11075.207} C_VEL
LIN {X 0,Y 404.707,Z 295.791,A -85,B 0,C 180,E1 -11075.577,E2 -11075.577} C_VEL
LIN {X 0,Y 401.523,Z 304.477,A -85,B 0,C 180,E1 -11076.045,E2 -11076.045} C_VEL
LIN {X 0,Y 400.618,Z 309.557,A -85,B 0,C 180,E1 -11076.416,E2 -11076.416} C_VEL
LIN {X 0,Y 399.786,Z 320.734,A -85,B 0,C 180,E1 -11077.449,E2 -11077.449} C_VEL
LIN {X 0,Y 399.044,Z 330.712,A -85,B 0,C 180,E1 -11078.61,E2 -11078.61} C_VEL
LIN {X 0,Y 398.253,Z 339.656,A -85,B 0,C 180,E1 -11079.882,E2 -11079.882} C_VEL
LIN {X 0,Y 397.579,Z 347.322,A -85,B 0,C 180,E1 -11081.212,E2 -11081.212} C_VEL
LIN {X 0,Y 396.991,Z 354.216,A -85,B 0,C 180,E1 -11082.677,E2 -11082.677} C_VEL
LIN {X 0,Y 396.484,Z 360.513,A -85,B 0,C 180,E1 -11084.369,E2 -11084.369} C_VEL
LIN {X 0,Y 396.179,Z 365.082,A -85,B 0,C 180,E1 -11085.96,E2 -11085.96} C_VEL
LIN {X 0,Y 395.899,Z 368.527,A -85,B 0,C 180,E1 -11087.565,E2 -11087.565} C_VEL
LIN {X 0,Y 395.791,Z 370.229,A -85,B 0,C 180,E1 -11088.64,E2 -11088.64} C_VEL
LIN {X 0,Y 395.715,Z 371.498,A -85,B 0,C 180,E1 -11089.733,E2 -11089.733} C_VEL
LIN {X 0,Y 395.639,Z 372.255,A -85,B 0,C 180,E1 -11090.81,E2 -11090.81} C_VEL
LIN {X 0,Y 395.636,Z 372.578,A -85,B 0,C 180,E1 -11092.527,E2 -11092.527} C_VEL
LIN {X 0,Y 395.671,Z 371.881,A -85,B 0,C 180,E1 -11094.113,E2 -11094.113} C_VEL
LIN {X 0,Y 395.796,Z 370.823,A -85,B 0,C 180,E1 -11095.224,E2 -11095.224} C_VEL
LIN {X 0,Y 396.004,Z 368.285,A -85,B 0,C 180,E1 -11096.908,E2 -11096.908} C_VEL
LIN {X 0,Y 396.318,Z 364.511,A -85,B 0,C 180,E1 -11098.607,E2 -11098.607} C_VEL
LIN {X 0,Y 396.743,Z 359.312,A -85,B 0,C 180,E1 -11100.322,E2 -11100.322} C_VEL
LIN {X 0,Y 397.31,Z 352.513,A -85,B 0,C 180,E1 -11102.051,E2 -11102.051} C_VEL
LIN {X 0,Y 397.936,Z 345.631,A -85,B 0,C 180,E1 -11103.446,E2 -11103.446} C_VEL
LIN {X 0,Y 398.786,Z 336.462,A -85,B 0,C 180,E1 -11104.943,E2 -11104.943} C_VEL
LIN {X 0,Y 399.711,Z 326.27,A -85,B 0,C 180,E1 -11106.275,E2 -11106.275} C_VEL
LIN {X 0,Y 400.592,Z 315.448,A -85,B 0,C 180,E1 -11107.406,E2 -11107.406} C_VEL
LIN {X 0,Y 401.426,Z 303.752,A -85,B 0,C 180,E1 -11108.363,E2 -11108.363} C_VEL
LIN {X 0,Y 402.146,Z 291.567,A -85,B 0,C 180,E1 -11109.128,E2 -11109.128} C_VEL
LIN {X 0,Y 402.615,Z 279.227,A -85,B 0,C 180,E1 -11109.693,E2 -11109.693} C_VEL
LIN {X 0,Y 402.997,Z 265.457,A -85,B 0,C 180,E1 -11110.089,E2 -11110.089} C_VEL
LIN {X 0,Y 404.249,Z 183.483,A -85,B 0,C 180,E1 -11111.583,E2 -11111.583} C_VEL
LIN {X 0,Y 399.677,Z 162.663,A -85,B 0,C 180,E1 -11112.236,E2 -11112.236} C_VEL
LIN {X 0,Y 399.545,Z 161.967,A -85,B 0,C 180,E1 -11112.295,E2 -11112.295} C_VEL
LIN {X 0,Y 398.36,Z 154.962,A -85,B 0,C 180,E1 -11114.036,E2 -11114.036} C_VEL
LIN {X 0,Y 397.159,Z 149.014,A -85,B 0,C 180,E1 -11115.59,E2 -11115.59} C_VEL
LIN {X 0,Y 397.116,Z 149.021,A -85,B 0,C 180,E1 -11119.096,E2 -11119.096} C_VEL
LIN {X 0,Y 397.106,Z 149.025,A -85,B 0,C 180,E1 -11121.727,E2 -11121.727} C_VEL
LIN {X 0,Y 397.123,Z 149.023,A -85,B 0,C 180,E1 -11125.508,E2 -11125.508} C_VEL
LIN {X 0,Y 397.076,Z 149.023,A -85,B 0,C 180,E1 -11129.119,E2 -11129.119} C_VEL
LIN {X 0,Y 397.192,Z 149.008,A -85,B 0,C 180,E1 -11132.611,E2 -11132.611} C_VEL
LIN {X 0,Y 397.132,Z 149.015,A -85,B 0,C 180,E1 -11135.983,E2 -11135.983} C_VEL
LIN {X 0,Y 397.138,Z 149.015,A -85,B 0,C 180,E1 -11139.706,E2 -11139.706} C_VEL
LIN {X 0,Y 397.181,Z 149.008,A -85,B 0,C 180,E1 -11142.846,E2 -11142.846} C_VEL
LIN {X 0,Y 397.229,Z 149,A -85,B 0,C 180,E1 -11146.704,E2 -11146.704} C_VEL
LIN {X 0,Y 397.217,Z 149.002,A -85,B 0,C 180,E1 -11149.81,E2 -11149.81} C_VEL
LIN {X 0,Y 397.32,Z 148.994,A -85,B 0,C 180,E1 -11152.888,E2 -11152.888} C_VEL
LIN {X 0,Y 397.246,Z 148.995,A -85,B 0,C 180,E1 -11154.926,E2 -11154.926} C_VEL
LIN {X 0,Y 397.448,Z 148.973,A -85,B 0,C 180,E1 -11157.974,E2 -11157.974} C_VEL
LIN {X 0,Y 397.574,Z 148.956,A -85,B 0,C 180,E1 -11160.001,E2 -11160.001} C_VEL
LIN {X 0,Y 397.327,Z 148.987,A -85,B 0,C 180,E1 -11163.043,E2 -11163.043} C_VEL
LIN {X 0,Y 397.333,Z 148.982,A -85,B 0,C 180,E1 -11166.093,E2 -11166.093} C_VEL
LIN {X 0,Y 397.236,Z 148.998,A -85,B 0,C 180,E1 -11169.163,E2 -11169.163} C_VEL
LIN {X 0,Y 397.221,Z 149.002,A -85,B 0,C 180,E1 -11172.259,E2 -11172.259} C_VEL
LIN {X 0,Y 397.128,Z 149.014,A -85,B 0,C 180,E1 -11175.395,E2 -11175.395} C_VEL
LIN {X 0,Y 397.153,Z 149.012,A -85,B 0,C 180,E1 -11178.575,E2 -11178.575} C_VEL
LIN {X 0,Y 397.095,Z 149.016,A -85,B 0,C 180,E1 -11181.819,E2 -11181.819} C_VEL
LIN {X 0,Y 397.105,Z 149.019,A -85,B 0,C 180,E1 -11185.136,E2 -11185.136} C_VEL
LIN {X 0,Y 397.063,Z 149.023,A -85,B 0,C 180,E1 -11188.549,E2 -11188.549} C_VEL
LIN {X 0,Y 397.077,Z 149.023,A -85,B 0,C 180,E1 -11191.835,E2 -11191.835} C_VEL
LIN {X 0,Y 397.117,Z 149.012,A -85,B 0,C 180,E1 -11194.495,E2 -11194.495} C_VEL
LIN {X 0,Y 397.088,Z 149.016,A -85,B 0,C 180,E1 -11198.278,E2 -11198.278} C_VEL
LIN {X 0,Y 397.048,Z 149.028,A -85,B 0,C 180,E1 -11200.915,E2 -11200.915} C_VEL
LIN {X 0,Y 397.089,Z 149.021,A -85,B 0,C 180,E1 -11203.651,E2 -11203.651} C_VEL
LIN {X 0,Y 397.093,Z 149.025,A -85,B 0,C 180,E1 -11206.523,E2 -11206.523} C_VEL
LIN {X 0,Y 397.088,Z 149.026,A -85,B 0,C 180,E1 -11210.42,E2 -11210.42} C_VEL
LIN {X 0,Y 397.098,Z 149.016,A -85,B 0,C 180,E1 -11213.005,E2 -11213.005} C_VEL
LIN {X 0,Y 397.101,Z 149.018,A -85,B 0,C 180,E1 -11216.287,E2 -11216.287} C_VEL
LIN {X 0,Y 397.08,Z 149.025,A -85,B 0,C 180,E1 -11219.118,E2 -11219.118} C_VEL
LIN {X 0,Y 397.155,Z 149.124,A -85,B 0,C 180,E1 -11221.351,E2 -11221.351} C_VEL
LIN {X 0,Y 399.983,Z 162.807,A -85,B 0,C 180,E1 -11224.502,E2 -11224.502} C_VEL
LIN {X 0,Y 400.534,Z 166.598,A -85,B 0,C 180,E1 -11225.337,E2 -11225.337} C_VEL
LIN {X 0,Y 399.482,Z 181.162,A -85,B 0,C 180,E1 -11228.319,E2 -11228.319} C_VEL
LIN {X 0,Y 398.978,Z 188.181,A -85,B 0,C 180,E1 -11229.741,E2 -11229.741} C_VEL
LIN {X 0,Y 403.329,Z 214.771,A -85,B 0,C 180,E1 -11230.491,E2 -11230.491} C_VEL
LIN {X 0,Y 403.742,Z 220.759,A -85,B 0,C 180,E1 -11230.627,E2 -11230.627} C_VEL
LIN {X 0,Y 402.728,Z 297.586,A -85,B 0,C 180,E1 -11232.054,E2 -11232.054} C_VEL
LIN {X 0,Y 401.999,Z 311.304,A -85,B 0,C 180,E1 -11232.514,E2 -11232.514} C_VEL
LIN {X 0,Y 401.269,Z 323.665,A -85,B 0,C 180,E1 -11233.137,E2 -11233.137} C_VEL
LIN {X 0,Y 400.436,Z 335.532,A -85,B 0,C 180,E1 -11233.953,E2 -11233.953} C_VEL
LIN {X 0,Y 399.48,Z 346.961,A -85,B 0,C 180,E1 -11234.96,E2 -11234.96} C_VEL
LIN {X 0,Y 398.666,Z 357.264,A -85,B 0,C 180,E1 -11236.1,E2 -11236.1} C_VEL
LIN {X 0,Y 397.963,Z 365.728,A -85,B 0,C 180,E1 -11237.247,E2 -11237.247} C_VEL
LIN {X 0,Y 397.058,Z 374.897,A -85,B 0,C 180,E1 -11238.773,E2 -11238.773} C_VEL
LIN {X 0,Y 396.518,Z 382.3,A -85,B 0,C 180,E1 -11240.306,E2 -11240.306} C_VEL
LIN {X 0,Y 396.163,Z 388.247,A -85,B 0,C 180,E1 -11241.841,E2 -11241.841} C_VEL
LIN {X 0,Y 395.898,Z 392.945,A -85,B 0,C 180,E1 -11243.375,E2 -11243.375} C_VEL
LIN {X 0,Y 395.83,Z 396.531,A -85,B 0,C 180,E1 -11244.907,E2 -11244.907} C_VEL
LIN {X 0,Y 395.775,Z 398.363,A -85,B 0,C 180,E1 -11245.927,E2 -11245.927} C_VEL
LIN {X 0,Y 395.805,Z 400.736,A -85,B 0,C 180,E1 -11247.965,E2 -11247.965} C_VEL
LIN {X 0,Y 395.813,Z 401.332,A -85,B 0,C 180,E1 -11248.983,E2 -11248.983} C_VEL
LIN {X 0,Y 395.802,Z 401.509,A -85,B 0,C 180,E1 -11250,E2 -11250} C_VEL
LIN {X 0,Y 395.813,Z 401.267,A -85,B 0,C 180,E1 -11251.018,E2 -11251.018} C_VEL
LIN {X 0,Y 395.806,Z 400.635,A -85,B 0,C 180,E1 -11252.035,E2 -11252.035} C_VEL
LIN {X 0,Y 395.734,Z 399.608,A -85,B 0,C 180,E1 -11253.054,E2 -11253.054} C_VEL
LIN {X 0,Y 395.775,Z 398.153,A -85,B 0,C 180,E1 -11254.073,E2 -11254.073} C_VEL
LIN {X 0,Y 395.802,Z 394.753,A -85,B 0,C 180,E1 -11255.767,E2 -11255.767} C_VEL
LIN {X 0,Y 396.064,Z 389.462,A -85,B 0,C 180,E1 -11257.648,E2 -11257.648} C_VEL
LIN {X 0,Y 396.361,Z 383.817,A -85,B 0,C 180,E1 -11259.183,E2 -11259.183} C_VEL
LIN {X 0,Y 396.827,Z 376.751,A -85,B 0,C 180,E1 -11260.717,E2 -11260.717} C_VEL
LIN {X 0,Y 397.61,Z 367.912,A -85,B 0,C 180,E1 -11262.246,E2 -11262.246} C_VEL
LIN {X 0,Y 398.277,Z 359.281,A -85,B 0,C 180,E1 -11263.465,E2 -11263.465} C_VEL
LIN {X 0,Y 399.083,Z 348.882,A -85,B 0,C 180,E1 -11264.664,E2 -11264.664} C_VEL
LIN {X 0,Y 399.908,Z 337.81,A -85,B 0,C 180,E1 -11265.677,E2 -11265.677} C_VEL
LIN {X 0,Y 400.801,Z 325.411,A -85,B 0,C 180,E1 -11266.556,E2 -11266.556} C_VEL
LIN {X 0,Y 401.498,Z 313.651,A -85,B 0,C 180,E1 -11267.181,E2 -11267.181} C_VEL
LIN {X 0,Y 402.143,Z 300.974,A -85,B 0,C 180,E1 -11267.645,E2 -11267.645} C_VEL
LIN {X 0,Y 402.484,Z 283.157,A -85,B 0,C 180,E1 -11268.023,E2 -11268.023} C_VEL
LIN {X 0,Y 403.115,Z 216.953,A -85,B 0,C 180,E1 -11269.23,E2 -11269.23} C_VEL
LIN {X 0,Y 398.79,Z 188.715,A -85,B 0,C 180,E1 -11269.996,E2 -11269.996} C_VEL
LIN {X 0,Y 399.98,Z 172.559,A -85,B 0,C 180,E1 -11273.288,E2 -11273.288} C_VEL
LIN {X 0,Y 400.421,Z 165.887,A -85,B 0,C 180,E1 -11274.664,E2 -11274.664} C_VEL
LIN {X 0,Y 398.189,Z 154.068,A -85,B 0,C 180,E1 -11277.316,E2 -11277.316} C_VEL
LIN {X 0,Y 397.154,Z 149.014,A -85,B 0,C 180,E1 -11278.494,E2 -11278.494} C_VEL
LIN {X 0,Y 397.082,Z 149.025,A -85,B 0,C 180,E1 -11282.072,E2 -11282.072} C_VEL
LIN {X 0,Y 397.12,Z 149.021,A -85,B 0,C 180,E1 -11285.502,E2 -11285.502} C_VEL
LIN {X 0,Y 397.098,Z 149.018,A -85,B 0,C 180,E1 -11288.855,E2 -11288.855} C_VEL
LIN {X 0,Y 397.059,Z 149.022,A -85,B 0,C 180,E1 -11292.269,E2 -11292.269} C_VEL
LIN {X 0,Y 397.09,Z 149.022,A -85,B 0,C 180,E1 -11295.069,E2 -11295.069} C_VEL
LIN {X 0,Y 397.057,Z 149.022,A -85,B 0,C 180,E1 -11298.023,E2 -11298.023} C_VEL
LIN {X 0,Y 397.098,Z 149.018,A -85,B 0,C 180,E1 -11301.724,E2 -11301.724} C_VEL
LIN {X 0,Y 397.122,Z 149.016,A -85,B 0,C 180,E1 -11305.506,E2 -11305.506} C_VEL
LIN {X 0,Y 397.081,Z 149.024,A -85,B 0,C 180,E1 -11309.117,E2 -11309.117} C_VEL
LIN {X 0,Y 397.096,Z 149.021,A -85,B 0,C 180,E1 -11312.602,E2 -11312.602} C_VEL
LIN {X 0,Y 397.117,Z 149.015,A -85,B 0,C 180,E1 -11315.98,E2 -11315.98} C_VEL
LIN {X 0,Y 397.144,Z 149.011,A -85,B 0,C 180,E1 -11319.704,E2 -11319.704} C_VEL
LIN {X 0,Y 397.158,Z 149.014,A -85,B 0,C 180,E1 -11322.858,E2 -11322.858} C_VEL
LIN {X 0,Y 397.234,Z 149.005,A -85,B 0,C 180,E1 -11326.702,E2 -11326.702} C_VEL
LIN {X 0,Y 397.217,Z 149.003,A -85,B 0,C 180,E1 -11329.808,E2 -11329.808} C_VEL
LIN {X 0,Y 397.298,Z 148.994,A -85,B 0,C 180,E1 -11332.886,E2 -11332.886} C_VEL
LIN {X 0,Y 397.236,Z 149.001,A -85,B 0,C 180,E1 -11334.924,E2 -11334.924} C_VEL
LIN {X 0,Y 397.444,Z 148.977,A -85,B 0,C 180,E1 -11337.972,E2 -11337.972} C_VEL
LIN {X 0,Y 397.325,Z 148.989,A -85,B 0,C 180,E1 -11341.013,E2 -11341.013} C_VEL
LIN {X 0,Y 397.324,Z 148.989,A -85,B 0,C 180,E1 -11343.041,E2 -11343.041} C_VEL
LIN {X 0,Y 397.298,Z 148.994,A -85,B 0,C 180,E1 -11346.483,E2 -11346.483} C_VEL
LIN {X 0,Y 397.23,Z 149.001,A -85,B 0,C 180,E1 -11349.161,E2 -11349.161} C_VEL
LIN {X 0,Y 397.217,Z 149.005,A -85,B 0,C 180,E1 -11352.257,E2 -11352.257} C_VEL
LIN {X 0,Y 397.124,Z 149.016,A -85,B 0,C 180,E1 -11355.393,E2 -11355.393} C_VEL
LIN {X 0,Y 397.094,Z 149.018,A -85,B 0,C 180,E1 -11358.576,E2 -11358.576} C_VEL
LIN {X 0,Y 397.091,Z 149.023,A -85,B 0,C 180,E1 -11361.818,E2 -11361.818} C_VEL
LIN {X 0,Y 397.103,Z 149.018,A -85,B 0,C 180,E1 -11365.134,E2 -11365.134} C_VEL
LIN {X 0,Y 397.062,Z 149.021,A -85,B 0,C 180,E1 -11368.547,E2 -11368.547} C_VEL
LIN {X 0,Y 397.079,Z 149.022,A -85,B 0,C 180,E1 -11371.835,E2 -11371.835} C_VEL
LIN {X 0,Y 397.118,Z 149.015,A -85,B 0,C 180,E1 -11374.493,E2 -11374.493} C_VEL
LIN {X 0,Y 397.088,Z 149.018,A -85,B 0,C 180,E1 -11378.275,E2 -11378.275} C_VEL
LIN {X 0,Y 397.048,Z 149.023,A -85,B 0,C 180,E1 -11381.975,E2 -11381.975} C_VEL
LIN {X 0,Y 397.082,Z 149.025,A -85,B 0,C 180,E1 -11385.068,E2 -11385.068} C_VEL
LIN {X 0,Y 397.048,Z 149.023,A -85,B 0,C 180,E1 -11388.023,E2 -11388.023} C_VEL
LIN {X 0,Y 397.089,Z 149.019,A -85,B 0,C 180,E1 -11391.723,E2 -11391.723} C_VEL
LIN {X 0,Y 397.112,Z 149.016,A -85,B 0,C 180,E1 -11395.505,E2 -11395.505} C_VEL
LIN {X 0,Y 397.07,Z 149.024,A -85,B 0,C 180,E1 -11399.116,E2 -11399.116} C_VEL
LIN {X 0,Y 397.056,Z 149.024,A -85,B 0,C 180,E1 -11402.251,E2 -11402.251} C_VEL
LIN {X 0,Y 397.096,Z 149.022,A -85,B 0,C 180,E1 -11404.864,E2 -11404.864} C_VEL
LIN {X 0,Y 397.087,Z 149.021,A -85,B 0,C 180,E1 -11408.181,E2 -11408.181} C_VEL
LIN {X 0,Y 397.103,Z 149.016,A -85,B 0,C 180,E1 -11411.423,E2 -11411.423} C_VEL
LIN {X 0,Y 397.116,Z 149.019,A -85,B 0,C 180,E1 -11414.605,E2 -11414.605} C_VEL
LIN {X 0,Y 397.206,Z 149.004,A -85,B 0,C 180,E1 -11417.741,E2 -11417.741} C_VEL
LIN {X 0,Y 397.219,Z 149.003,A -85,B 0,C 180,E1 -11420.837,E2 -11420.837} C_VEL
LIN {X 0,Y 397.319,Z 148.993,A -85,B 0,C 180,E1 -11423.907,E2 -11423.907} C_VEL
LIN {X 0,Y 397.431,Z 148.981,A -85,B 0,C 180,E1 -11427.973,E2 -11427.973} C_VEL
LIN {X 0,Y 397.312,Z 149.105,A -85,B 0,C 180,E1 -11428.955,E2 -11428.955} C_VEL
LIN {X 0,Y 398.772,Z 157.227,A -85,B 0,C 180,E1 -11431.01,E2 -11431.01} C_VEL
LIN {X 0,Y 399.143,Z 161.749,A -85,B 0,C 180,E1 -11432.112,E2 -11432.112} C_VEL
LIN {X 0,Y 403.637,Z 184.057,A -85,B 0,C 180,E1 -11432.756,E2 -11432.756} C_VEL
LIN {X 0,Y 402.371,Z 269.553,A -85,B 0,C 180,E1 -11434.326,E2 -11434.326} C_VEL
LIN {X 0,Y 401.904,Z 282.665,A -85,B 0,C 180,E1 -11434.77,E2 -11434.77} C_VEL
LIN {X 0,Y 401.396,Z 295.173,A -85,B 0,C 180,E1 -11435.4,E2 -11435.4} C_VEL
LIN {X 0,Y 400.788,Z 306.436,A -85,B 0,C 180,E1 -11436.166,E2 -11436.166} C_VEL
LIN {X 0,Y 400.618,Z 309.557,A -85,B 0,C 180,E1 -11436.416,E2 -11436.416} C_VEL
LIN {X 0,Y 399.674,Z 314.646,A -85,B 0,C 180,E1 -11436.825,E2 -11436.825} C_VEL
LIN {X 0,Y 396.266,Z 322.66,A -85,B 0,C 180,E1 -11437.512,E2 -11437.512} C_VEL
LIN {X 0,Y 392.805,Z 330.194,A -85,B 0,C 180,E1 -11438.303,E2 -11438.303} C_VEL
LIN {X 0,Y 391.789,Z 334.531,A -85,B 0,C 180,E1 -11438.869,E2 -11438.869} C_VEL
LIN {X 0,Y 390.888,Z 343.943,A -85,B 0,C 180,E1 -11440.358,E2 -11440.358} C_VEL
LIN {X 0,Y 390.196,Z 352.016,A -85,B 0,C 180,E1 -11441.954,E2 -11441.954} C_VEL
LIN {X 0,Y 389.641,Z 358.443,A -85,B 0,C 180,E1 -11443.561,E2 -11443.561} C_VEL
LIN {X 0,Y 389.231,Z 363.539,A -85,B 0,C 180,E1 -11445.178,E2 -11445.178} C_VEL
LIN {X 0,Y 388.926,Z 367.455,A -85,B 0,C 180,E1 -11446.805,E2 -11446.805} C_VEL
LIN {X 0,Y 388.778,Z 369.471,A -85,B 0,C 180,E1 -11447.897,E2 -11447.897} C_VEL
LIN {X 0,Y 388.607,Z 371.892,A -85,B 0,C 180,E1 -11449.88,E2 -11449.88} C_VEL
LIN {X 0,Y 388.537,Z 372.705,A -85,B 0,C 180,E1 -11451.209,E2 -11451.209} C_VEL
LIN {X 0,Y 388.543,Z 372.815,A -85,B 0,C 180,E1 -11452.71,E2 -11452.71} C_VEL
LIN {X 0,Y 388.622,Z 371.829,A -85,B 0,C 180,E1 -11454.579,E2 -11454.579} C_VEL
LIN {X 0,Y 388.74,Z 370.566,A -85,B 0,C 180,E1 -11455.715,E2 -11455.715} C_VEL
LIN {X 0,Y 389.068,Z 367.109,A -85,B 0,C 180,E1 -11457.736,E2 -11457.736} C_VEL
LIN {X 0,Y 389.429,Z 362.442,A -85,B 0,C 180,E1 -11459.587,E2 -11459.587} C_VEL
LIN {X 0,Y 389.937,Z 356.991,A -85,B 0,C 180,E1 -11461.21,E2 -11461.21} C_VEL
LIN {X 0,Y 390.641,Z 349.436,A -85,B 0,C 180,E1 -11462.972,E2 -11462.972} C_VEL
LIN {X 0,Y 391.372,Z 342.279,A -85,B 0,C 180,E1 -11464.308,E2 -11464.308} C_VEL
LIN {X 0,Y 392.177,Z 333.75,A -85,B 0,C 180,E1 -11465.621,E2 -11465.621} C_VEL
LIN {X 0,Y 393.094,Z 323.195,A -85,B 0,C 180,E1 -11466.927,E2 -11466.927} C_VEL
LIN {X 0,Y 394.026,Z 312.584,A -85,B 0,C 180,E1 -11467.977,E2 -11467.977} C_VEL
LIN {X 0,Y 394.899,Z 301.395,A -85,B 0,C 180,E1 -11468.854,E2 -11468.854} C_VEL
LIN {X 0,Y 395.515,Z 288.826,A -85,B 0,C 180,E1 -11469.604,E2 -11469.604} C_VEL
LIN {X 0,Y 396.014,Z 275.183,A -85,B 0,C 180,E1 -11470.174,E2 -11470.174} C_VEL
LIN {X 0,Y 396.408,Z 261.574,A -85,B 0,C 180,E1 -11470.504,E2 -11470.504} C_VEL
LIN {X 0,Y 397.612,Z 184.569,A -85,B 0,C 180,E1 -11471.927,E2 -11471.927} C_VEL
LIN {X 0,Y 393.462,Z 165.362,A -85,B 0,C 180,E1 -11472.542,E2 -11472.542} C_VEL
LIN {X 0,Y 392.536,Z 162.307,A -85,B 0,C 180,E1 -11472.679,E2 -11472.679} C_VEL
LIN {X 0,Y 390.46,Z 151.629,A -85,B 0,C 180,E1 -11475.416,E2 -11475.416} C_VEL
LIN {X 0,Y 390.113,Z 149.893,A -85,B 0,C 180,E1 -11475.891,E2 -11475.891} C_VEL
LIN {X 0,Y 390.079,Z 149.898,A -85,B 0,C 180,E1 -11479.175,E2 -11479.175} C_VEL
LIN {X 0,Y 390.043,Z 149.904,A -85,B 0,C 180,E1 -11482.449,E2 -11482.449} C_VEL
LIN {X 0,Y 390.065,Z 149.897,A -85,B 0,C 180,E1 -11486.046,E2 -11486.046} C_VEL
LIN {X 0,Y 390.044,Z 149.897,A -85,B 0,C 180,E1 -11489.87,E2 -11489.87} C_VEL
LIN {X 0,Y 390.112,Z 149.892,A -85,B 0,C 180,E1 -11493.233,E2 -11493.233} C_VEL
LIN {X 0,Y 390.105,Z 149.891,A -85,B 0,C 180,E1 -11496.751,E2 -11496.751} C_VEL
LIN {X 0,Y 390.102,Z 149.891,A -85,B 0,C 180,E1 -11499.984,E2 -11499.984} C_VEL
LIN {X 0,Y 390.138,Z 149.886,A -85,B 0,C 180,E1 -11503.249,E2 -11503.249} C_VEL
LIN {X 0,Y 390.195,Z 149.877,A -85,B 0,C 180,E1 -11506.562,E2 -11506.562} C_VEL
LIN {X 0,Y 390.168,Z 149.881,A -85,B 0,C 180,E1 -11509.624,E2 -11509.624} C_VEL
LIN {X 0,Y 390.269,Z 149.871,A -85,B 0,C 180,E1 -11512.759,E2 -11512.759} C_VEL
LIN {X 0,Y 390.217,Z 149.871,A -85,B 0,C 180,E1 -11514.834,E2 -11514.834} C_VEL
LIN {X 0,Y 390.417,Z 149.848,A -85,B 0,C 180,E1 -11517.938,E2 -11517.938} C_VEL
LIN {X 0,Y 390.544,Z 149.831,A -85,B 0,C 180,E1 -11520.001,E2 -11520.001} C_VEL
LIN {X 0,Y 390.264,Z 149.867,A -85,B 0,C 180,E1 -11523.098,E2 -11523.098} C_VEL
LIN {X 0,Y 390.287,Z 149.859,A -85,B 0,C 180,E1 -11526.203,E2 -11526.203} C_VEL
LIN {X 0,Y 390.194,Z 149.876,A -85,B 0,C 180,E1 -11529.33,E2 -11529.33} C_VEL
LIN {X 0,Y 390.173,Z 149.882,A -85,B 0,C 180,E1 -11532.484,E2 -11532.484} C_VEL
LIN {X 0,Y 390.07,Z 149.891,A -85,B 0,C 180,E1 -11535.68,E2 -11535.68} C_VEL
LIN {X 0,Y 390.095,Z 149.891,A -85,B 0,C 180,E1 -11538.923,E2 -11538.923} C_VEL
LIN {X 0,Y 390.036,Z 149.897,A -85,B 0,C 180,E1 -11542.235,E2 -11542.235} C_VEL
LIN {X 0,Y 390.052,Z 149.892,A -85,B 0,C 180,E1 -11545.723,E2 -11545.723} C_VEL
LIN {X 0,Y 390.024,Z 149.903,A -85,B 0,C 180,E1 -11549.113,E2 -11549.113} C_VEL
LIN {X 0,Y 390.04,Z 149.899,A -85,B 0,C 180,E1 -11552.723,E2 -11552.723} C_VEL
LIN {X 0,Y 390.042,Z 149.899,A -85,B 0,C 180,E1 -11555.822,E2 -11555.822} C_VEL
LIN {X 0,Y 390.035,Z 149.903,A -85,B 0,C 180,E1 -11559.212,E2 -11559.212} C_VEL
LIN {X 0,Y 390.031,Z 149.902,A -85,B 0,C 180,E1 -11562.372,E2 -11562.372} C_VEL
LIN {X 0,Y 390.043,Z 149.904,A -85,B 0,C 180,E1 -11565.354,E2 -11565.354} C_VEL
LIN {X 0,Y 390.017,Z 149.906,A -85,B 0,C 180,E1 -11568.185,E2 -11568.185} C_VEL
LIN {X 0,Y 390.06,Z 149.899,A -85,B 0,C 180,E1 -11570.904,E2 -11570.904} C_VEL
LIN {X 0,Y 390.084,Z 149.897,A -85,B 0,C 180,E1 -11574.793,E2 -11574.793} C_VEL
LIN {X 0,Y 390.025,Z 149.901,A -85,B 0,C 180,E1 -11578.496,E2 -11578.496} C_VEL
LIN {X 0,Y 390.133,Z 150.095,A -85,B 0,C 180,E1 -11581.037,E2 -11581.037} C_VEL
LIN {X 0,Y 392.813,Z 162.848,A -85,B 0,C 180,E1 -11584.046,E2 -11584.046} C_VEL
LIN {X 0,Y 393.625,Z 167.904,A -85,B 0,C 180,E1 -11585.192,E2 -11585.192} C_VEL
LIN {X 0,Y 392.45,Z 183.245,A -85,B 0,C 180,E1 -11588.386,E2 -11588.386} C_VEL
LIN {X 0,Y 392.109,Z 187.922,A -85,B 0,C 180,E1 -11589.351,E2 -11589.351} C_VEL
LIN {X 0,Y 396.532,Z 214.696,A -85,B 0,C 180,E1 -11590.126,E2 -11590.126} C_VEL
LIN {X 0,Y 397.102,Z 219.996,A -85,B 0,C 180,E1 -11590.26,E2 -11590.26} C_VEL
LIN {X 0,Y 396.046,Z 296.726,A -85,B 0,C 180,E1 -11591.707,E2 -11591.707} C_VEL
LIN {X 0,Y 395.34,Z 309.867,A -85,B 0,C 180,E1 -11592.142,E2 -11592.142} C_VEL
LIN {X 0,Y 394.538,Z 322.546,A -85,B 0,C 180,E1 -11592.774,E2 -11592.774} C_VEL
LIN {X 0,Y 393.742,Z 333.854,A -85,B 0,C 180,E1 -11593.539,E2 -11593.539} C_VEL
LIN {X 0,Y 392.705,Z 345.539,A -85,B 0,C 180,E1 -11594.561,E2 -11594.561} C_VEL
LIN {X 0,Y 391.838,Z 356.378,A -85,B 0,C 180,E1 -11595.761,E2 -11595.761} C_VEL
LIN {X 0,Y 391.018,Z 365.558,A -85,B 0,C 180,E1 -11597.017,E2 -11597.017} C_VEL
LIN {X 0,Y 390.074,Z 374.709,A -85,B 0,C 180,E1 -11598.569,E2 -11598.569} C_VEL
LIN {X 0,Y 389.473,Z 382.099,A -85,B 0,C 180,E1 -11600.129,E2 -11600.129} C_VEL
LIN {X 0,Y 389.108,Z 388.036,A -85,B 0,C 180,E1 -11601.692,E2 -11601.692} C_VEL
LIN {X 0,Y 388.827,Z 392.723,A -85,B 0,C 180,E1 -11603.253,E2 -11603.253} C_VEL
LIN {X 0,Y 388.725,Z 396.3,A -85,B 0,C 180,E1 -11604.814,E2 -11604.814} C_VEL
LIN {X 0,Y 388.698,Z 398.124,A -85,B 0,C 180,E1 -11605.853,E2 -11605.853} C_VEL
LIN {X 0,Y 388.703,Z 400.487,A -85,B 0,C 180,E1 -11607.928,E2 -11607.928} C_VEL
LIN {X 0,Y 388.742,Z 401.08,A -85,B 0,C 180,E1 -11608.964,E2 -11608.964} C_VEL
LIN {X 0,Y 388.73,Z 401.248,A -85,B 0,C 180,E1 -11610,E2 -11610} C_VEL
LIN {X 0,Y 388.742,Z 401.001,A -85,B 0,C 180,E1 -11611.036,E2 -11611.036} C_VEL
LIN {X 0,Y 388.704,Z 400.364,A -85,B 0,C 180,E1 -11612.073,E2 -11612.073} C_VEL
LIN {X 0,Y 388.641,Z 399.332,A -85,B 0,C 180,E1 -11613.11,E2 -11613.11} C_VEL
LIN {X 0,Y 388.699,Z 397.867,A -85,B 0,C 180,E1 -11614.148,E2 -11614.148} C_VEL
LIN {X 0,Y 388.753,Z 393.877,A -85,B 0,C 180,E1 -11616.112,E2 -11616.112} C_VEL
LIN {X 0,Y 388.996,Z 389.149,A -85,B 0,C 180,E1 -11617.788,E2 -11617.788} C_VEL
LIN {X 0,Y 389.415,Z 382.404,A -85,B 0,C 180,E1 -11619.61,E2 -11619.61} C_VEL
LIN {X 0,Y 389.902,Z 375.032,A -85,B 0,C 180,E1 -11621.173,E2 -11621.173} C_VEL
LIN {X 0,Y 390.803,Z 365.899,A -85,B 0,C 180,E1 -11622.727,E2 -11622.727} C_VEL
LIN {X 0,Y 391.589,Z 355.814,A -85,B 0,C 180,E1 -11624.094,E2 -11624.094} C_VEL
LIN {X 0,Y 392.456,Z 344.564,A -85,B 0,C 180,E1 -11625.316,E2 -11625.316} C_VEL
LIN {X 0,Y 393.304,Z 334.147,A -85,B 0,C 180,E1 -11626.213,E2 -11626.213} C_VEL
LIN {X 0,Y 394.229,Z 321.642,A -85,B 0,C 180,E1 -11627.04,E2 -11627.04} C_VEL
LIN {X 0,Y 394.933,Z 309.231,A -85,B 0,C 180,E1 -11627.643,E2 -11627.643} C_VEL
LIN {X 0,Y 395.457,Z 296.66,A -85,B 0,C 180,E1 -11628.053,E2 -11628.053} C_VEL
LIN {X 0,Y 396.389,Z 217.845,A -85,B 0,C 180,E1 -11629.53,E2 -11629.53} C_VEL
LIN {X 0,Y 391.905,Z 188.586,A -85,B 0,C 180,E1 -11630.318,E2 -11630.318} C_VEL
LIN {X 0,Y 393.285,Z 170.902,A -85,B 0,C 180,E1 -11633.988,E2 -11633.988} C_VEL
LIN {X 0,Y 393.461,Z 166.976,A -85,B 0,C 180,E1 -11634.819,E2 -11634.819} C_VEL
LIN {X 0,Y 390.888,Z 153.684,A -85,B 0,C 180,E1 -11637.871,E2 -11637.871} C_VEL
LIN {X 0,Y 390.108,Z 149.892,A -85,B 0,C 180,E1 -11638.77,E2 -11638.77} C_VEL
LIN {X 0,Y 390.046,Z 149.897,A -85,B 0,C 180,E1 -11642.722,E2 -11642.722} C_VEL
LIN {X 0,Y 390.058,Z 149.897,A -85,B 0,C 180,E1 -11645.825,E2 -11645.825} C_VEL
LIN {X 0,Y 390.042,Z 149.9,A -85,B 0,C 180,E1 -11649.212,E2 -11649.212} C_VEL
LIN {X 0,Y 390.034,Z 149.897,A -85,B 0,C 180,E1 -11652.372,E2 -11652.372} C_VEL
LIN {X 0,Y 390.045,Z 149.902,A -85,B 0,C 180,E1 -11655.354,E2 -11655.354} C_VEL
LIN {X 0,Y 390.02,Z 149.899,A -85,B 0,C 180,E1 -11658.184,E2 -11658.184} C_VEL
LIN {X 0,Y 390.064,Z 149.897,A -85,B 0,C 180,E1 -11660.904,E2 -11660.904} C_VEL
LIN {X 0,Y 390.075,Z 149.895,A -85,B 0,C 180,E1 -11664.791,E2 -11664.791} C_VEL
LIN {X 0,Y 390.026,Z 149.9,A -85,B 0,C 180,E1 -11668.495,E2 -11668.495} C_VEL
LIN {X 0,Y 390.033,Z 149.897,A -85,B 0,C 180,E1 -11672.063,E2 -11672.063} C_VEL
LIN {X 0,Y 390.048,Z 149.896,A -85,B 0,C 180,E1 -11675.516,E2 -11675.516} C_VEL
LIN {X 0,Y 390.06,Z 149.899,A -85,B 0,C 180,E1 -11678.877,E2 -11678.877} C_VEL
LIN {X 0,Y 390.073,Z 149.894,A -85,B 0,C 180,E1 -11682.163,E2 -11682.163} C_VEL
LIN {X 0,Y 390.099,Z 149.889,A -85,B 0,C 180,E1 -11685.39,E2 -11685.39} C_VEL
LIN {X 0,Y 390.176,Z 149.879,A -85,B 0,C 180,E1 -11687.516,E2 -11687.516} C_VEL
LIN {X 0,Y 390.194,Z 149.881,A -85,B 0,C 180,E1 -11690.67,E2 -11690.67} C_VEL
LIN {X 0,Y 390.287,Z 149.867,A -85,B 0,C 180,E1 -11693.797,E2 -11693.797} C_VEL
LIN {X 0,Y 390.411,Z 149.853,A -85,B 0,C 180,E1 -11697.936,E2 -11697.936} C_VEL
LIN {X 0,Y 390.295,Z 149.865,A -85,B 0,C 180,E1 -11701.031,E2 -11701.031} C_VEL
LIN {X 0,Y 390.26,Z 149.869,A -85,B 0,C 180,E1 -11703.096,E2 -11703.096} C_VEL
LIN {X 0,Y 390.258,Z 149.871,A -85,B 0,C 180,E1 -11706.475,E2 -11706.475} C_VEL
LIN {X 0,Y 390.188,Z 149.878,A -85,B 0,C 180,E1 -11709.328,E2 -11709.328} C_VEL
LIN {X 0,Y 390.197,Z 149.879,A -85,B 0,C 180,E1 -11713.437,E2 -11713.437} C_VEL
LIN {X 0,Y 390.074,Z 149.893,A -85,B 0,C 180,E1 -11717.27,E2 -11717.27} C_VEL
LIN {X 0,Y 390.07,Z 149.893,A -85,B 0,C 180,E1 -11720.461,E2 -11720.461} C_VEL
LIN {X 0,Y 390.057,Z 149.897,A -85,B 0,C 180,E1 -11723.352,E2 -11723.352} C_VEL
LIN {X 0,Y 390.03,Z 149.898,A -85,B 0,C 180,E1 -11726.773,E2 -11726.773} C_VEL
LIN {X 0,Y 390.035,Z 149.897,A -85,B 0,C 180,E1 -11730.299,E2 -11730.299} C_VEL
LIN {X 0,Y 390.067,Z 149.894,A -85,B 0,C 180,E1 -11734.023,E2 -11734.023} C_VEL
LIN {X 0,Y 390.037,Z 149.901,A -85,B 0,C 180,E1 -11737.549,E2 -11737.549} C_VEL
LIN {X 0,Y 390.013,Z 149.902,A -85,B 0,C 180,E1 -11740.813,E2 -11740.813} C_VEL
LIN {X 0,Y 390.041,Z 149.897,A -85,B 0,C 180,E1 -11743.883,E2 -11743.883} C_VEL
LIN {X 0,Y 390.043,Z 149.899,A -85,B 0,C 180,E1 -11746.787,E2 -11746.787} C_VEL
LIN {X 0,Y 390.005,Z 149.902,A -85,B 0,C 180,E1 -11749.554,E2 -11749.554} C_VEL
LIN {X 0,Y 390.035,Z 149.898,A -85,B 0,C 180,E1 -11752.449,E2 -11752.449} C_VEL
LIN {X 0,Y 390.056,Z 149.894,A -85,B 0,C 180,E1 -11756.044,E2 -11756.044} C_VEL
LIN {X 0,Y 390.037,Z 149.897,A -85,B 0,C 180,E1 -11759.869,E2 -11759.869} C_VEL
LIN {X 0,Y 390.024,Z 149.9,A -85,B 0,C 180,E1 -11763.225,E2 -11763.225} C_VEL
LIN {X 0,Y 390.052,Z 149.9,A -85,B 0,C 180,E1 -11766.766,E2 -11766.766} C_VEL
LIN {X 0,Y 390.078,Z 149.893,A -85,B 0,C 180,E1 -11769.981,E2 -11769.981} C_VEL
LIN {X 0,Y 390.098,Z 149.889,A -85,B 0,C 180,E1 -11773.246,E2 -11773.246} C_VEL
LIN {X 0,Y 390.188,Z 149.882,A -85,B 0,C 180,E1 -11776.561,E2 -11776.561} C_VEL
LIN {X 0,Y 390.178,Z 149.882,A -85,B 0,C 180,E1 -11780.67,E2 -11780.67} C_VEL
LIN {X 0,Y 390.274,Z 149.87,A -85,B 0,C 180,E1 -11783.797,E2 -11783.797} C_VEL
LIN {X 0,Y 390.399,Z 149.857,A -85,B 0,C 180,E1 -11787.936,E2 -11787.936} C_VEL
LIN {X 0,Y 390.309,Z 150,A -85,B 0,C 180,E1 -11788.71,E2 -11788.71} C_VEL
LIN {X 0,Y 391.908,Z 159.035,A -85,B 0,C 180,E1 -11791.027,E2 -11791.027} C_VEL
LIN {X 0,Y 392.263,Z 162.111,A -85,B 0,C 180,E1 -11791.769,E2 -11791.769} C_VEL
LIN {X 0,Y 396.902,Z 184.777,A -85,B 0,C 180,E1 -11792.442,E2 -11792.442} C_VEL
LIN {X 0,Y 395.613,Z 269.587,A -85,B 0,C 180,E1 -11794.025,E2 -11794.025} C_VEL
LIN {X 0,Y 395.149,Z 282.291,A -85,B 0,C 180,E1 -11794.456,E2 -11794.456} C_VEL
LIN {X 0,Y 394.599,Z 295.184,A -85,B 0,C 180,E1 -11795.109,E2 -11795.109} C_VEL
LIN {X 0,Y 393.94,Z 306.534,A -85,B 0,C 180,E1 -11795.888,E2 -11795.888} C_VEL
LIN {X 0,Y 393.129,Z 318.267,A -85,B 0,C 180,E1 -11796.931,E2 -11796.931} C_VEL
LIN {X 0,Y 392.271,Z 328.846,A -85,B 0,C 180,E1 -11798.111,E2 -11798.111} C_VEL
LIN {X 0,Y 391.789,Z 334.531,A -85,B 0,C 180,E1 -11798.869,E2 -11798.869} C_VEL
LIN {X 0,Y 390.793,Z 338.72,A -85,B 0,C 180,E1 -11799.467,E2 -11799.467} C_VEL
LIN {X 0,Y 387.381,Z 345.179,A -85,B 0,C 180,E1 -11800.459,E2 -11800.459} C_VEL
LIN {X 0,Y 383.978,Z 351.029,A -85,B 0,C 180,E1 -11801.535,E2 -11801.535} C_VEL
LIN {X 0,Y 383.006,Z 354.256,A -85,B 0,C 180,E1 -11802.256,E2 -11802.256} C_VEL
LIN {X 0,Y 382.477,Z 360.063,A -85,B 0,C 180,E1 -11803.82,E2 -11803.82} C_VEL
LIN {X 0,Y 382.116,Z 364.87,A -85,B 0,C 180,E1 -11805.467,E2 -11805.467} C_VEL
LIN {X 0,Y 381.788,Z 368.522,A -85,B 0,C 180,E1 -11807.129,E2 -11807.129} C_VEL
LIN {X 0,Y 381.652,Z 370.324,A -85,B 0,C 180,E1 -11808.243,E2 -11808.243} C_VEL
LIN {X 0,Y 381.515,Z 372.289,A -85,B 0,C 180,E1 -11810.038,E2 -11810.038} C_VEL
LIN {X 0,Y 381.428,Z 373.065,A -85,B 0,C 180,E1 -11811.624,E2 -11811.624} C_VEL
LIN {X 0,Y 381.463,Z 373.053,A -85,B 0,C 180,E1 -11812.902,E2 -11812.902} C_VEL
LIN {X 0,Y 381.503,Z 372.632,A -85,B 0,C 180,E1 -11813.909,E2 -11813.909} C_VEL
LIN {X 0,Y 381.644,Z 371.173,A -85,B 0,C 180,E1 -11815.535,E2 -11815.535} C_VEL
LIN {X 0,Y 381.914,Z 368.301,A -85,B 0,C 180,E1 -11817.39,E2 -11817.39} C_VEL
LIN {X 0,Y 382.256,Z 364.303,A -85,B 0,C 180,E1 -11819.158,E2 -11819.158} C_VEL
LIN {X 0,Y 382.778,Z 358.896,A -85,B 0,C 180,E1 -11820.937,E2 -11820.937} C_VEL
LIN {X 0,Y 383.389,Z 352.753,A -85,B 0,C 180,E1 -11822.519,E2 -11822.519} C_VEL
LIN {X 0,Y 384.089,Z 346.016,A -85,B 0,C 180,E1 -11823.923,E2 -11823.923} C_VEL
LIN {X 0,Y 385.012,Z 337.088,A -85,B 0,C 180,E1 -11825.431,E2 -11825.431} C_VEL
LIN {X 0,Y 385.947,Z 327.377,A -85,B 0,C 180,E1 -11826.754,E2 -11826.754} C_VEL
LIN {X 0,Y 386.988,Z 316.274,A -85,B 0,C 180,E1 -11827.966,E2 -11827.966} C_VEL
LIN {X 0,Y 387.807,Z 305.565,A -85,B 0,C 180,E1 -11828.89,E2 -11828.89} C_VEL
LIN {X 0,Y 388.592,Z 293.555,A -85,B 0,C 180,E1 -11829.692,E2 -11829.692} C_VEL
LIN {X 0,Y 389.206,Z 280.403,A -85,B 0,C 180,E1 -11830.334,E2 -11830.334} C_VEL
LIN {X 0,Y 389.607,Z 267.857,A -85,B 0,C 180,E1 -11830.726,E2 -11830.726} C_VEL
LIN {X 0,Y 390.917,Z 184.981,A -85,B 0,C 180,E1 -11832.301,E2 -11832.301} C_VEL
LIN {X 0,Y 386.904,Z 166.932,A -85,B 0,C 180,E1 -11832.902,E2 -11832.902} C_VEL
LIN {X 0,Y 385.5,Z 162.614,A -85,B 0,C 180,E1 -11833.088,E2 -11833.088} C_VEL
LIN {X 0,Y 383.068,Z 150.769,A -85,B 0,C 180,E1 -11836.258,E2 -11836.258} C_VEL
LIN {X 0,Y 383.04,Z 150.773,A -85,B 0,C 180,E1 -11838.787,E2 -11838.787} C_VEL
LIN {X 0,Y 383,Z 150.784,A -85,B 0,C 180,E1 -11842.096,E2 -11842.096} C_VEL
LIN {X 0,Y 383.015,Z 150.779,A -85,B 0,C 180,E1 -11845.333,E2 -11845.333} C_VEL
LIN {X 0,Y 382.98,Z 150.779,A -85,B 0,C 180,E1 -11849.082,E2 -11849.082} C_VEL
LIN {X 0,Y 383.055,Z 150.769,A -85,B 0,C 180,E1 -11852.699,E2 -11852.699} C_VEL
LIN {X 0,Y 383.032,Z 150.771,A -85,B 0,C 180,E1 -11856.194,E2 -11856.194} C_VEL
LIN {X 0,Y 383.054,Z 150.77,A -85,B 0,C 180,E1 -11859.599,E2 -11859.599} C_VEL
LIN {X 0,Y 383.093,Z 150.762,A -85,B 0,C 180,E1 -11862.932,E2 -11862.932} C_VEL
LIN {X 0,Y 383.125,Z 150.757,A -85,B 0,C 180,E1 -11866.465,E2 -11866.465} C_VEL
LIN {X 0,Y 383.144,Z 150.755,A -85,B 0,C 180,E1 -11870.499,E2 -11870.499} C_VEL
LIN {X 0,Y 383.257,Z 150.741,A -85,B 0,C 180,E1 -11873.684,E2 -11873.684} C_VEL
LIN {X 0,Y 383.384,Z 150.724,A -85,B 0,C 180,E1 -11877.9,E2 -11877.9} C_VEL
LIN {X 0,Y 383.513,Z 150.707,A -85,B 0,C 180,E1 -11880.001,E2 -11880.001} C_VEL
LIN {X 0,Y 383.202,Z 150.746,A -85,B 0,C 180,E1 -11883.155,E2 -11883.155} C_VEL
LIN {X 0,Y 383.243,Z 150.737,A -85,B 0,C 180,E1 -11886.318,E2 -11886.318} C_VEL
LIN {X 0,Y 383.144,Z 150.755,A -85,B 0,C 180,E1 -11889.503,E2 -11889.503} C_VEL
LIN {X 0,Y 383.128,Z 150.759,A -85,B 0,C 180,E1 -11893.537,E2 -11893.537} C_VEL
LIN {X 0,Y 383.06,Z 150.762,A -85,B 0,C 180,E1 -11897.437,E2 -11897.437} C_VEL
LIN {X 0,Y 383.019,Z 150.768,A -85,B 0,C 180,E1 -11900.642,E2 -11900.642} C_VEL
LIN {X 0,Y 383.01,Z 150.777,A -85,B 0,C 180,E1 -11903.81,E2 -11903.81} C_VEL
LIN {X 0,Y 382.97,Z 150.776,A -85,B 0,C 180,E1 -11907.309,E2 -11907.309} C_VEL
LIN {X 0,Y 382.98,Z 150.772,A -85,B 0,C 180,E1 -11910.92,E2 -11910.92} C_VEL
LIN {X 0,Y 383.013,Z 150.769,A -85,B 0,C 180,E1 -11914.669,E2 -11914.669} C_VEL
LIN {X 0,Y 382.992,Z 150.773,A -85,B 0,C 180,E1 -11917.902,E2 -11917.902} C_VEL
LIN {X 0,Y 382.962,Z 150.782,A -85,B 0,C 180,E1 -11921.351,E2 -11921.351} C_VEL
LIN {X 0,Y 382.991,Z 150.777,A -85,B 0,C 180,E1 -11924.303,E2 -11924.303} C_VEL
LIN {X 0,Y 382.984,Z 150.784,A -85,B 0,C 180,E1 -11927.237,E2 -11927.237} C_VEL
LIN {X 0,Y 382.988,Z 150.783,A -85,B 0,C 180,E1 -11930.419,E2 -11930.419} C_VEL
LIN {X 0,Y 383.025,Z 150.77,A -85,B 0,C 180,E1 -11934.044,E2 -11934.044} C_VEL
LIN {X 0,Y 382.989,Z 150.779,A -85,B 0,C 180,E1 -11937.579,E2 -11937.579} C_VEL
LIN {X 0,Y 383.035,Z 150.82,A -85,B 0,C 180,E1 -11940.644,E2 -11940.644} C_VEL
LIN {X 0,Y 385.751,Z 163.488,A -85,B 0,C 180,E1 -11943.71,E2 -11943.71} C_VEL
LIN {X 0,Y 386.702,Z 169.066,A -85,B 0,C 180,E1 -11945.004,E2 -11945.004} C_VEL
LIN {X 0,Y 385.719,Z 182.135,A -85,B 0,C 180,E1 -11947.786,E2 -11947.786} C_VEL
LIN {X 0,Y 385.249,Z 187.57,A -85,B 0,C 180,E1 -11948.926,E2 -11948.926} C_VEL
LIN {X 0,Y 389.621,Z 213.447,A -85,B 0,C 180,E1 -11949.716,E2 -11949.716} C_VEL
LIN {X 0,Y 390.463,Z 220.832,A -85,B 0,C 180,E1 -11949.91,E2 -11949.91} C_VEL
LIN {X 0,Y 389.322,Z 297.139,A -85,B 0,C 180,E1 -11951.38,E2 -11951.38} C_VEL
LIN {X 0,Y 388.545,Z 310.812,A -85,B 0,C 180,E1 -11951.853,E2 -11951.853} C_VEL
LIN {X 0,Y 387.703,Z 323.653,A -85,B 0,C 180,E1 -11952.529,E2 -11952.529} C_VEL
LIN {X 0,Y 386.801,Z 335.396,A -85,B 0,C 180,E1 -11953.371,E2 -11953.371} C_VEL
LIN {X 0,Y 385.74,Z 346.741,A -85,B 0,C 180,E1 -11954.411,E2 -11954.411} C_VEL
LIN {X 0,Y 384.859,Z 357.063,A -85,B 0,C 180,E1 -11955.603,E2 -11955.603} C_VEL
LIN {X 0,Y 384.077,Z 365.391,A -85,B 0,C 180,E1 -11956.778,E2 -11956.778} C_VEL
LIN {X 0,Y 383.104,Z 374.522,A -85,B 0,C 180,E1 -11958.358,E2 -11958.358} C_VEL
LIN {X 0,Y 382.454,Z 381.899,A -85,B 0,C 180,E1 -11959.946,E2 -11959.946} C_VEL
LIN {X 0,Y 382.043,Z 387.825,A -85,B 0,C 180,E1 -11961.537,E2 -11961.537} C_VEL
LIN {X 0,Y 381.748,Z 392.502,A -85,B 0,C 180,E1 -11963.127,E2 -11963.127} C_VEL
LIN {X 0,Y 381.628,Z 396.07,A -85,B 0,C 180,E1 -11964.717,E2 -11964.717} C_VEL
LIN {X 0,Y 381.623,Z 397.885,A -85,B 0,C 180,E1 -11965.776,E2 -11965.776} C_VEL
LIN {X 0,Y 381.6,Z 400.238,A -85,B 0,C 180,E1 -11967.889,E2 -11967.889} C_VEL
LIN {X 0,Y 381.655,Z 400.828,A -85,B 0,C 180,E1 -11968.945,E2 -11968.945} C_VEL
LIN {X 0,Y 381.661,Z 400.987,A -85,B 0,C 180,E1 -11970,E2 -11970} C_VEL
LIN {X 0,Y 381.673,Z 400.735,A -85,B 0,C 180,E1 -11971.055,E2 -11971.055} C_VEL
LIN {X 0,Y 381.602,Z 400.091,A -85,B 0,C 180,E1 -11972.111,E2 -11972.111} C_VEL
LIN {X 0,Y 381.552,Z 399.055,A -85,B 0,C 180,E1 -11973.168,E2 -11973.168} C_VEL
LIN {X 0,Y 381.623,Z 397.579,A -85,B 0,C 180,E1 -11974.225,E2 -11974.225} C_VEL
LIN {X 0,Y 381.656,Z 393.943,A -85,B 0,C 180,E1 -11976.071,E2 -11976.071} C_VEL
LIN {X 0,Y 381.92,Z 388.835,A -85,B 0,C 180,E1 -11977.933,E2 -11977.933} C_VEL
LIN {X 0,Y 382.365,Z 382.067,A -85,B 0,C 180,E1 -11979.789,E2 -11979.789} C_VEL
LIN {X 0,Y 382.904,Z 374.68,A -85,B 0,C 180,E1 -11981.38,E2 -11981.38} C_VEL
LIN {X 0,Y 383.831,Z 365.521,A -85,B 0,C 180,E1 -11982.962,E2 -11982.962} C_VEL
LIN {X 0,Y 384.592,Z 356.32,A -85,B 0,C 180,E1 -11984.241,E2 -11984.241} C_VEL
LIN {X 0,Y 385.469,Z 345.42,A -85,B 0,C 180,E1 -11985.465,E2 -11985.465} C_VEL
LIN {X 0,Y 386.46,Z 333.652,A -85,B 0,C 180,E1 -11986.508,E2 -11986.508} C_VEL
LIN {X 0,Y 387.42,Z 321.063,A -85,B 0,C 180,E1 -11987.349,E2 -11987.349} C_VEL
LIN {X 0,Y 388.192,Z 307.781,A -85,B 0,C 180,E1 -11987.994,E2 -11987.994} C_VEL
LIN {X 0,Y 388.68,Z 295.638,A -85,B 0,C 180,E1 -11988.379,E2 -11988.379} C_VEL
LIN {X 0,Y 389.699,Z 218.884,A -85,B 0,C 180,E1 -11989.836,E2 -11989.836} C_VEL
LIN {X 0,Y 384.984,Z 188.228,A -85,B 0,C 180,E1 -11990.7,E2 -11990.7} C_VEL
LIN {X 0,Y 386.346,Z 172.046,A -85,B 0,C 180,E1 -11994.12,E2 -11994.12} C_VEL
LIN {X 0,Y 386.478,Z 167.929,A -85,B 0,C 180,E1 -11995.012,E2 -11995.012} C_VEL
LIN {X 0,Y 384.155,Z 155.955,A -85,B 0,C 180,E1 -11997.809,E2 -11997.809} C_VEL
LIN {X 0,Y 383.033,Z 150.776,A -85,B 0,C 180,E1 -11999.093,E2 -11999.093} C_VEL
LIN {X 0,Y 382.99,Z 150.778,A -85,B 0,C 180,E1 -12002.422,E2 -12002.422} C_VEL
LIN {X 0,Y 383.027,Z 150.772,A -85,B 0,C 180,E1 -12005.956,E2 -12005.956} C_VEL
LIN {X 0,Y 382.99,Z 150.779,A -85,B 0,C 180,E1 -12009.581,E2 -12009.581} C_VEL
LIN {X 0,Y 383.011,Z 150.773,A -85,B 0,C 180,E1 -12012.778,E2 -12012.778} C_VEL
LIN {X 0,Y 382.995,Z 150.776,A -85,B 0,C 180,E1 -12015.788,E2 -12015.788} C_VEL
LIN {X 0,Y 382.966,Z 150.78,A -85,B 0,C 180,E1 -12018.8,E2 -12018.8} C_VEL
LIN {X 0,Y 382.999,Z 150.773,A -85,B 0,C 180,E1 -12022.097,E2 -12022.097} C_VEL
LIN {X 0,Y 383.016,Z 150.775,A -85,B 0,C 180,E1 -12025.331,E2 -12025.331} C_VEL
LIN {X 0,Y 382.986,Z 150.78,A -85,B 0,C 180,E1 -12029.081,E2 -12029.081} C_VEL
LIN {X 0,Y 382.99,Z 150.779,A -85,B 0,C 180,E1 -12032.692,E2 -12032.692} C_VEL
LIN {X 0,Y 383.015,Z 150.772,A -85,B 0,C 180,E1 -12036.191,E2 -12036.191} C_VEL
LIN {X 0,Y 383.061,Z 150.766,A -85,B 0,C 180,E1 -12039.598,E2 -12039.598} C_VEL
LIN {X 0,Y 383.075,Z 150.767,A -85,B 0,C 180,E1 -12042.929,E2 -12042.929} C_VEL
LIN {X 0,Y 383.131,Z 150.763,A -85,B 0,C 180,E1 -12046.463,E2 -12046.463} C_VEL
LIN {X 0,Y 383.145,Z 150.761,A -85,B 0,C 180,E1 -12050.497,E2 -12050.497} C_VEL
LIN {X 0,Y 383.243,Z 150.743,A -85,B 0,C 180,E1 -12053.682,E2 -12053.682} C_VEL
LIN {X 0,Y 383.377,Z 150.729,A -85,B 0,C 180,E1 -12057.898,E2 -12057.898} C_VEL
LIN {X 0,Y 383.266,Z 150.74,A -85,B 0,C 180,E1 -12061.05,E2 -12061.05} C_VEL
LIN {X 0,Y 383.376,Z 150.732,A -85,B 0,C 180,E1 -12062.1,E2 -12062.1} C_VEL
LIN {X 0,Y 383.224,Z 150.748,A -85,B 0,C 180,E1 -12066.463,E2 -12066.463} C_VEL
LIN {X 0,Y 383.139,Z 150.758,A -85,B 0,C 180,E1 -12069.501,E2 -12069.501} C_VEL
LIN {X 0,Y 383.128,Z 150.76,A -85,B 0,C 180,E1 -12073.535,E2 -12073.535} C_VEL
LIN {X 0,Y 383.027,Z 150.772,A -85,B 0,C 180,E1 -12077.42,E2 -12077.42} C_VEL
LIN {X 0,Y 383.014,Z 150.771,A -85,B 0,C 180,E1 -12080.639,E2 -12080.639} C_VEL
LIN {X 0,Y 383.008,Z 150.777,A -85,B 0,C 180,E1 -12083.808,E2 -12083.808} C_VEL
LIN {X 0,Y 382.969,Z 150.781,A -85,B 0,C 180,E1 -12087.308,E2 -12087.308} C_VEL
LIN {X 0,Y 382.98,Z 150.777,A -85,B 0,C 180,E1 -12090.918,E2 -12090.918} C_VEL
LIN {X 0,Y 383.015,Z 150.772,A -85,B 0,C 180,E1 -12094.667,E2 -12094.667} C_VEL
LIN {X 0,Y 382.991,Z 150.775,A -85,B 0,C 180,E1 -12097.901,E2 -12097.901} C_VEL
LIN {X 0,Y 382.957,Z 150.784,A -85,B 0,C 180,E1 -12101.349,E2 -12101.349} C_VEL
LIN {X 0,Y 382.986,Z 150.775,A -85,B 0,C 180,E1 -12104.301,E2 -12104.301} C_VEL
LIN {X 0,Y 383.007,Z 150.777,A -85,B 0,C 180,E1 -12107.239,E2 -12107.239} C_VEL
LIN {X 0,Y 382.982,Z 150.777,A -85,B 0,C 180,E1 -12110.418,E2 -12110.418} C_VEL
LIN {X 0,Y 383.01,Z 150.772,A -85,B 0,C 180,E1 -12114.042,E2 -12114.042} C_VEL
LIN {X 0,Y 382.979,Z 150.776,A -85,B 0,C 180,E1 -12117.578,E2 -12117.578} C_VEL
LIN {X 0,Y 382.969,Z 150.779,A -85,B 0,C 180,E1 -12120.298,E2 -12120.298} C_VEL
LIN {X 0,Y 382.996,Z 150.775,A -85,B 0,C 180,E1 -12124.044,E2 -12124.044} C_VEL
LIN {X 0,Y 382.979,Z 150.776,A -85,B 0,C 180,E1 -12127.333,E2 -12127.333} C_VEL
LIN {X 0,Y 383.025,Z 150.775,A -85,B 0,C 180,E1 -12130.714,E2 -12130.714} C_VEL
LIN {X 0,Y 383.012,Z 150.774,A -85,B 0,C 180,E1 -12134.023,E2 -12134.023} C_VEL
LIN {X 0,Y 383.127,Z 150.757,A -85,B 0,C 180,E1 -12137.283,E2 -12137.283} C_VEL
LIN {X 0,Y 383.129,Z 150.761,A -85,B 0,C 180,E1 -12140.497,E2 -12140.497} C_VEL
LIN {X 0,Y 383.23,Z 150.746,A -85,B 0,C 180,E1 -12143.683,E2 -12143.683} C_VEL
LIN {X 0,Y 383.283,Z 150.745,A -85,B 0,C 180,E1 -12148.292,E2 -12148.292} C_VEL
LIN {X 0,Y 383.284,Z 150.786,A -85,B 0,C 180,E1 -12148.424,E2 -12148.424} C_VEL
LIN {X 0,Y 385.034,Z 160.858,A -85,B 0,C 180,E1 -12151.046,E2 -12151.046} C_VEL
LIN {X 0,Y 385.254,Z 162.187,A -85,B 0,C 180,E1 -12151.388,E2 -12151.388} C_VEL
LIN {X 0,Y 390.056,Z 184.457,A -85,B 0,C 180,E1 -12152.091,E2 -12152.091} C_VEL
LIN {X 0,Y 389.483,Z 231.753,A -85,B 0,C 180,E1 -12152.982,E2 -12152.982} C_VEL
LIN {X 0,Y 388.834,Z 270.018,A -85,B 0,C 180,E1 -12153.724,E2 -12153.724} C_VEL
LIN {X 0,Y 388.344,Z 283.003,A -85,B 0,C 180,E1 -12154.177,E2 -12154.177} C_VEL
LIN {X 0,Y 387.767,Z 295.887,A -85,B 0,C 180,E1 -12154.848,E2 -12154.848} C_VEL
LIN {X 0,Y 387.017,Z 308.215,A -85,B 0,C 180,E1 -12155.732,E2 -12155.732} C_VEL
LIN {X 0,Y 386.158,Z 319.704,A -85,B 0,C 180,E1 -12156.794,E2 -12156.794} C_VEL
LIN {X 0,Y 385.291,Z 330.036,A -85,B 0,C 180,E1 -12157.995,E2 -12157.995} C_VEL
LIN {X 0,Y 384.342,Z 340.169,A -85,B 0,C 180,E1 -12159.472,E2 -12159.472} C_VEL
LIN {X 0,Y 383.602,Z 347.703,A -85,B 0,C 180,E1 -12160.824,E2 -12160.824} C_VEL
LIN {X 0,Y 383.006,Z 354.256,A -85,B 0,C 180,E1 -12162.256,E2 -12162.256} C_VEL
LIN {X 0,Y 382.074,Z 357.306,A -85,B 0,C 180,E1 -12163.001,E2 -12163.001} C_VEL
LIN {X 0,Y 378.85,Z 361.822,A -85,B 0,C 180,E1 -12164.241,E2 -12164.241} C_VEL
LIN {X 0,Y 375.672,Z 365.596,A -85,B 0,C 180,E1 -12165.551,E2 -12165.551} C_VEL
LIN {X 0,Y 374.83,Z 367.486,A -85,B 0,C 180,E1 -12166.399,E2 -12166.399} C_VEL
LIN {X 0,Y 374.64,Z 369.473,A -85,B 0,C 180,E1 -12167.466,E2 -12167.466} C_VEL
LIN {X 0,Y 374.509,Z 371.146,A -85,B 0,C 180,E1 -12168.604,E2 -12168.604} C_VEL
LIN {X 0,Y 374.415,Z 372.683,A -85,B 0,C 180,E1 -12170.197,E2 -12170.197} C_VEL
LIN {X 0,Y 374.34,Z 373.393,A -85,B 0,C 180,E1 -12172.054,E2 -12172.054} C_VEL
LIN {X 0,Y 374.398,Z 373.227,A -85,B 0,C 180,E1 -12173.216,E2 -12173.216} C_VEL
LIN {X 0,Y 374.443,Z 372.584,A -85,B 0,C 180,E1 -12174.388,E2 -12174.388} C_VEL
LIN {X 0,Y 374.571,Z 371.254,A -85,B 0,C 180,E1 -12175.764,E2 -12175.764} C_VEL
LIN {X 0,Y 374.837,Z 368.879,A -85,B 0,C 180,E1 -12177.346,E2 -12177.346} C_VEL
LIN {X 0,Y 375.175,Z 364.997,A -85,B 0,C 180,E1 -12179.147,E2 -12179.147} C_VEL
LIN {X 0,Y 375.744,Z 359.452,A -85,B 0,C 180,E1 -12181.037,E2 -12181.037} C_VEL
LIN {X 0,Y 376.474,Z 352.511,A -85,B 0,C 180,E1 -12182.856,E2 -12182.856} C_VEL
LIN {X 0,Y 377.236,Z 345.562,A -85,B 0,C 180,E1 -12184.303,E2 -12184.303} C_VEL
LIN {X 0,Y 378.221,Z 336.518,A -85,B 0,C 180,E1 -12185.826,E2 -12185.826} C_VEL
LIN {X 0,Y 379.211,Z 326.697,A -85,B 0,C 180,E1 -12187.164,E2 -12187.164} C_VEL
LIN {X 0,Y 380.197,Z 316.704,A -85,B 0,C 180,E1 -12188.262,E2 -12188.262} C_VEL
LIN {X 0,Y 381.095,Z 305.544,A -85,B 0,C 180,E1 -12189.238,E2 -12189.238} C_VEL
LIN {X 0,Y 381.947,Z 292.805,A -85,B 0,C 180,E1 -12190.092,E2 -12190.092} C_VEL
LIN {X 0,Y 382.549,Z 280.105,A -85,B 0,C 180,E1 -12190.707,E2 -12190.707} C_VEL
LIN {X 0,Y 382.951,Z 267.341,A -85,B 0,C 180,E1 -12191.102,E2 -12191.102} C_VEL
LIN {X 0,Y 384.289,Z 185.963,A -85,B 0,C 180,E1 -12192.675,E2 -12192.675} C_VEL
LIN {X 0,Y 380.575,Z 169.194,A -85,B 0,C 180,E1 -12193.25,E2 -12193.25} C_VEL
LIN {X 0,Y 378.348,Z 162.917,A -85,B 0,C 180,E1 -12193.531,E2 -12193.531} C_VEL
LIN {X 0,Y 376.026,Z 151.645,A -85,B 0,C 180,E1 -12196.6,E2 -12196.6} C_VEL
LIN {X 0,Y 375.995,Z 151.653,A -85,B 0,C 180,E1 -12200.028,E2 -12200.028} C_VEL
LIN {X 0,Y 375.962,Z 151.66,A -85,B 0,C 180,E1 -12203.496,E2 -12203.496} C_VEL
LIN {X 0,Y 375.957,Z 151.655,A -85,B 0,C 180,E1 -12205.89,E2 -12205.89} C_VEL
LIN {X 0,Y 375.962,Z 151.653,A -85,B 0,C 180,E1 -12209.688,E2 -12209.688} C_VEL
LIN {X 0,Y 375.994,Z 151.649,A -85,B 0,C 180,E1 -12212.142,E2 -12212.142} C_VEL
LIN {X 0,Y 376.005,Z 151.649,A -85,B 0,C 180,E1 -12214.54,E2 -12214.54} C_VEL
LIN {X 0,Y 375.962,Z 151.653,A -85,B 0,C 180,E1 -12218.047,E2 -12218.047} C_VEL
LIN {X 0,Y 376.002,Z 151.648,A -85,B 0,C 180,E1 -12221.474,E2 -12221.474} C_VEL
LIN {X 0,Y 376.058,Z 151.644,A -85,B 0,C 180,E1 -12224.834,E2 -12224.834} C_VEL
LIN {X 0,Y 376.05,Z 151.639,A -85,B 0,C 180,E1 -12228.138,E2 -12228.138} C_VEL
LIN {X 0,Y 376.174,Z 151.619,A -85,B 0,C 180,E1 -12231.969,E2 -12231.969} C_VEL
LIN {X 0,Y 376.16,Z 151.624,A -85,B 0,C 180,E1 -12234.641,E2 -12234.641} C_VEL
LIN {X 0,Y 376.35,Z 151.6,A -85,B 0,C 180,E1 -12237.861,E2 -12237.861} C_VEL
LIN {X 0,Y 376.483,Z 151.582,A -85,B 0,C 180,E1 -12240.001,E2 -12240.001} C_VEL
LIN {X 0,Y 376.34,Z 151.599,A -85,B 0,C 180,E1 -12242.141,E2 -12242.141} C_VEL
LIN {X 0,Y 376.202,Z 151.615,A -85,B 0,C 180,E1 -12246.437,E2 -12246.437} C_VEL
LIN {X 0,Y 376.115,Z 151.632,A -85,B 0,C 180,E1 -12249.682,E2 -12249.682} C_VEL
LIN {X 0,Y 376.092,Z 151.637,A -85,B 0,C 180,E1 -12253.658,E2 -12253.658} C_VEL
LIN {X 0,Y 376.014,Z 151.641,A -85,B 0,C 180,E1 -12257.592,E2 -12257.592} C_VEL
LIN {X 0,Y 375.981,Z 151.644,A -85,B 0,C 180,E1 -12260.833,E2 -12260.833} C_VEL
LIN {X 0,Y 375.937,Z 151.654,A -85,B 0,C 180,E1 -12264.286,E2 -12264.286} C_VEL
LIN {X 0,Y 375.913,Z 151.651,A -85,B 0,C 180,E1 -12266.661,E2 -12266.661} C_VEL
LIN {X 0,Y 375.914,Z 151.66,A -85,B 0,C 180,E1 -12269.085,E2 -12269.085} C_VEL
LIN {X 0,Y 375.955,Z 151.653,A -85,B 0,C 180,E1 -12271.563,E2 -12271.563} C_VEL
LIN {X 0,Y 375.95,Z 151.654,A -85,B 0,C 180,E1 -12275.417,E2 -12275.417} C_VEL
LIN {X 0,Y 375.934,Z 151.652,A -85,B 0,C 180,E1 -12278.263,E2 -12278.263} C_VEL
LIN {X 0,Y 375.915,Z 151.661,A -85,B 0,C 180,E1 -12281.597,E2 -12281.597} C_VEL
LIN {X 0,Y 375.923,Z 151.661,A -85,B 0,C 180,E1 -12284.731,E2 -12284.731} C_VEL
LIN {X 0,Y 375.91,Z 151.663,A -85,B 0,C 180,E1 -12287.697,E2 -12287.697} C_VEL
LIN {X 0,Y 375.937,Z 151.66,A -85,B 0,C 180,E1 -12290.534,E2 -12290.534} C_VEL
LIN {X 0,Y 375.964,Z 151.647,A -85,B 0,C 180,E1 -12293.497,E2 -12293.497} C_VEL
LIN {X 0,Y 375.962,Z 151.651,A -85,B 0,C 180,E1 -12295.889,E2 -12295.889} C_VEL
LIN {X 0,Y 375.967,Z 151.654,A -85,B 0,C 180,E1 -12299.688,E2 -12299.688} C_VEL
LIN {X 0,Y 375.993,Z 151.838,A -85,B 0,C 180,E1 -12300.308,E2 -12300.308} C_VEL
LIN {X 0,Y 378.566,Z 163.721,A -85,B 0,C 180,E1 -12303.259,E2 -12303.259} C_VEL
LIN {X 0,Y 379.779,Z 170.23,A -85,B 0,C 180,E1 -12304.81,E2 -12304.81} C_VEL
LIN {X 0,Y 378.907,Z 181.991,A -85,B 0,C 180,E1 -12307.365,E2 -12307.365} C_VEL
LIN {X 0,Y 378.37,Z 187.353,A -85,B 0,C 180,E1 -12308.51,E2 -12308.51} C_VEL
LIN {X 0,Y 382.745,Z 212.391,A -85,B 0,C 180,E1 -12309.295,E2 -12309.295} C_VEL
LIN {X 0,Y 383.839,Z 221.672,A -85,B 0,C 180,E1 -12309.548,E2 -12309.548} C_VEL
LIN {X 0,Y 382.648,Z 296.422,A -85,B 0,C 180,E1 -12311.008,E2 -12311.008} C_VEL
LIN {X 0,Y 381.86,Z 310.239,A -85,B 0,C 180,E1 -12311.49,E2 -12311.49} C_VEL
LIN {X 0,Y 381.008,Z 322.667,A -85,B 0,C 180,E1 -12312.142,E2 -12312.142} C_VEL
LIN {X 0,Y 380.014,Z 335.365,A -85,B 0,C 180,E1 -12313.065,E2 -12313.065} C_VEL
LIN {X 0,Y 378.895,Z 346.667,A -85,B 0,C 180,E1 -12314.122,E2 -12314.122} C_VEL
LIN {X 0,Y 377.949,Z 356.944,A -85,B 0,C 180,E1 -12315.334,E2 -12315.334} C_VEL
LIN {X 0,Y 376.983,Z 366.888,A -85,B 0,C 180,E1 -12316.799,E2 -12316.799} C_VEL
LIN {X 0,Y 375.96,Z 375.721,A -85,B 0,C 180,E1 -12318.407,E2 -12318.407} C_VEL
LIN {X 0,Y 375.327,Z 382.793,A -85,B 0,C 180,E1 -12320.026,E2 -12320.026} C_VEL
LIN {X 0,Y 374.865,Z 389.28,A -85,B 0,C 180,E1 -12321.917,E2 -12321.917} C_VEL
LIN {X 0,Y 374.626,Z 393.562,A -85,B 0,C 180,E1 -12323.537,E2 -12323.537} C_VEL
LIN {X 0,Y 374.536,Z 395.84,A -85,B 0,C 180,E1 -12324.617,E2 -12324.617} C_VEL
LIN {X 0,Y 374.548,Z 397.646,A -85,B 0,C 180,E1 -12325.696,E2 -12325.696} C_VEL
LIN {X 0,Y 374.499,Z 399.99,A -85,B 0,C 180,E1 -12327.849,E2 -12327.849} C_VEL
LIN {X 0,Y 374.57,Z 400.575,A -85,B 0,C 180,E1 -12328.925,E2 -12328.925} C_VEL
LIN {X 0,Y 374.593,Z 400.726,A -85,B 0,C 180,E1 -12330,E2 -12330} C_VEL
LIN {X 0,Y 374.586,Z 400.469,A -85,B 0,C 180,E1 -12331.075,E2 -12331.075} C_VEL
LIN {X 0,Y 374.466,Z 398.778,A -85,B 0,C 180,E1 -12333.228,E2 -12333.228} C_VEL
LIN {X 0,Y 374.548,Z 397.292,A -85,B 0,C 180,E1 -12334.305,E2 -12334.305} C_VEL
LIN {X 0,Y 374.552,Z 394.03,A -85,B 0,C 180,E1 -12336.019,E2 -12336.019} C_VEL
LIN {X 0,Y 374.767,Z 390.149,A -85,B 0,C 180,E1 -12337.543,E2 -12337.543} C_VEL
LIN {X 0,Y 375.155,Z 383.849,A -85,B 0,C 180,E1 -12339.435,E2 -12339.435} C_VEL
LIN {X 0,Y 375.687,Z 376.987,A -85,B 0,C 180,E1 -12341.055,E2 -12341.055} C_VEL
LIN {X 0,Y 376.548,Z 368.434,A -85,B 0,C 180,E1 -12342.669,E2 -12342.669} C_VEL
LIN {X 0,Y 377.368,Z 359.627,A -85,B 0,C 180,E1 -12344.011,E2 -12344.011} C_VEL
LIN {X 0,Y 378.156,Z 349.96,A -85,B 0,C 180,E1 -12345.219,E2 -12345.219} C_VEL
LIN {X 0,Y 379.096,Z 339.409,A -85,B 0,C 180,E1 -12346.284,E2 -12346.284} C_VEL
LIN {X 0,Y 380.071,Z 327.741,A -85,B 0,C 180,E1 -12347.209,E2 -12347.209} C_VEL
LIN {X 0,Y 380.891,Z 315.621,A -85,B 0,C 180,E1 -12347.934,E2 -12347.934} C_VEL
LIN {X 0,Y 381.679,Z 302.478,A -85,B 0,C 180,E1 -12348.485,E2 -12348.485} C_VEL
LIN {X 0,Y 382.056,Z 289.828,A -85,B 0,C 180,E1 -12348.814,E2 -12348.814} C_VEL
LIN {X 0,Y 382.914,Z 219.169,A -85,B 0,C 180,E1 -12350.169,E2 -12350.169} C_VEL
LIN {X 0,Y 378.085,Z 187.982,A -85,B 0,C 180,E1 -12351.072,E2 -12351.072} C_VEL
LIN {X 0,Y 379.477,Z 172.246,A -85,B 0,C 180,E1 -12354.459,E2 -12354.459} C_VEL
LIN {X 0,Y 379.47,Z 168.863,A -85,B 0,C 180,E1 -12355.213,E2 -12355.213} C_VEL
LIN {X 0,Y 376.907,Z 155.987,A -85,B 0,C 180,E1 -12358.293,E2 -12358.293} C_VEL
LIN {X 0,Y 375.979,Z 151.655,A -85,B 0,C 180,E1 -12359.386,E2 -12359.386} C_VEL
LIN {X 0,Y 375.953,Z 151.653,A -85,B 0,C 180,E1 -12362.829,E2 -12362.829} C_VEL
LIN {X 0,Y 375.96,Z 151.655,A -85,B 0,C 180,E1 -12365.416,E2 -12365.416} C_VEL
LIN {X 0,Y 375.94,Z 151.653,A -85,B 0,C 180,E1 -12368.263,E2 -12368.263} C_VEL
LIN {X 0,Y 375.92,Z 151.659,A -85,B 0,C 180,E1 -12371.597,E2 -12371.597} C_VEL
LIN {X 0,Y 375.925,Z 151.656,A -85,B 0,C 180,E1 -12374.73,E2 -12374.73} C_VEL
LIN {X 0,Y 375.93,Z 151.656,A -85,B 0,C 180,E1 -12377.699,E2 -12377.699} C_VEL
LIN {X 0,Y 375.94,Z 151.653,A -85,B 0,C 180,E1 -12380.534,E2 -12380.534} C_VEL
LIN {X 0,Y 375.963,Z 151.652,A -85,B 0,C 180,E1 -12383.496,E2 -12383.496} C_VEL
LIN {X 0,Y 375.962,Z 151.65,A -85,B 0,C 180,E1 -12385.888,E2 -12385.888} C_VEL
LIN {X 0,Y 375.966,Z 151.65,A -85,B 0,C 180,E1 -12389.687,E2 -12389.687} C_VEL
LIN {X 0,Y 375.933,Z 151.654,A -85,B 0,C 180,E1 -12392.135,E2 -12392.135} C_VEL
LIN {X 0,Y 375.973,Z 151.649,A -85,B 0,C 180,E1 -12395.716,E2 -12395.716} C_VEL
LIN {X 0,Y 375.985,Z 151.649,A -85,B 0,C 180,E1 -12399.196,E2 -12399.196} C_VEL
LIN {X 0,Y 376.014,Z 151.65,A -85,B 0,C 180,E1 -12402.598,E2 -12402.598} C_VEL
LIN {X 0,Y 376.095,Z 151.638,A -85,B 0,C 180,E1 -12406.342,E2 -12406.342} C_VEL
LIN {X 0,Y 376.116,Z 151.636,A -85,B 0,C 180,E1 -12410.318,E2 -12410.318} C_VEL
LIN {X 0,Y 376.202,Z 151.62,A -85,B 0,C 180,E1 -12413.563,E2 -12413.563} C_VEL
LIN {X 0,Y 376.342,Z 151.605,A -85,B 0,C 180,E1 -12417.859,E2 -12417.859} C_VEL
LIN {X 0,Y 376.237,Z 151.616,A -85,B 0,C 180,E1 -12421.069,E2 -12421.069} C_VEL
LIN {X 0,Y 376.341,Z 151.609,A -85,B 0,C 180,E1 -12422.14,E2 -12422.14} C_VEL
LIN {X 0,Y 376.195,Z 151.624,A -85,B 0,C 180,E1 -12426.447,E2 -12426.447} C_VEL
LIN {X 0,Y 376.11,Z 151.635,A -85,B 0,C 180,E1 -12429.681,E2 -12429.681} C_VEL
LIN {X 0,Y 376.092,Z 151.638,A -85,B 0,C 180,E1 -12433.656,E2 -12433.656} C_VEL
LIN {X 0,Y 375.985,Z 151.651,A -85,B 0,C 180,E1 -12437.577,E2 -12437.577} C_VEL
LIN {X 0,Y 375.98,Z 151.648,A -85,B 0,C 180,E1 -12440.831,E2 -12440.831} C_VEL
LIN {X 0,Y 375.935,Z 151.654,A -85,B 0,C 180,E1 -12444.284,E2 -12444.284} C_VEL
LIN {X 0,Y 375.911,Z 151.656,A -85,B 0,C 180,E1 -12446.659,E2 -12446.659} C_VEL
LIN {X 0,Y 375.913,Z 151.658,A -85,B 0,C 180,E1 -12449.083,E2 -12449.083} C_VEL
LIN {X 0,Y 375.955,Z 151.656,A -85,B 0,C 180,E1 -12451.561,E2 -12451.561} C_VEL
LIN {X 0,Y 375.954,Z 151.657,A -85,B 0,C 180,E1 -12455.415,E2 -12455.415} C_VEL
LIN {X 0,Y 375.932,Z 151.654,A -85,B 0,C 180,E1 -12458.262,E2 -12458.262} C_VEL
LIN {X 0,Y 375.912,Z 151.659,A -85,B 0,C 180,E1 -12461.596,E2 -12461.596} C_VEL
LIN {X 0,Y 375.917,Z 151.658,A -85,B 0,C 180,E1 -12464.729,E2 -12464.729} C_VEL
LIN {X 0,Y 375.921,Z 151.656,A -85,B 0,C 180,E1 -12467.698,E2 -12467.698} C_VEL
LIN {X 0,Y 375.931,Z 151.656,A -85,B 0,C 180,E1 -12470.533,E2 -12470.533} C_VEL
LIN {X 0,Y 375.954,Z 151.652,A -85,B 0,C 180,E1 -12473.496,E2 -12473.496} C_VEL
LIN {X 0,Y 375.952,Z 151.651,A -85,B 0,C 180,E1 -12475.887,E2 -12475.887} C_VEL
LIN {X 0,Y 375.955,Z 151.651,A -85,B 0,C 180,E1 -12479.686,E2 -12479.686} C_VEL
LIN {X 0,Y 375.911,Z 151.657,A -85,B 0,C 180,E1 -12482.134,E2 -12482.134} C_VEL
LIN {X 0,Y 375.93,Z 151.659,A -85,B 0,C 180,E1 -12484.533,E2 -12484.533} C_VEL
LIN {X 0,Y 375.964,Z 151.653,A -85,B 0,C 180,E1 -12486.886,E2 -12486.886} C_VEL
LIN {X 0,Y 375.967,Z 151.654,A -85,B 0,C 180,E1 -12490.337,E2 -12490.337} C_VEL
LIN {X 0,Y 375.967,Z 151.65,A -85,B 0,C 180,E1 -12493.716,E2 -12493.716} C_VEL
LIN {X 0,Y 376.095,Z 151.634,A -85,B 0,C 180,E1 -12497.041,E2 -12497.041} C_VEL
LIN {X 0,Y 376.099,Z 151.639,A -85,B 0,C 180,E1 -12500.318,E2 -12500.318} C_VEL
LIN {X 0,Y 376.189,Z 151.622,A -85,B 0,C 180,E1 -12503.564,E2 -12503.564} C_VEL
LIN {X 0,Y 376.295,Z 151.699,A -85,B 0,C 180,E1 -12508.16,E2 -12508.16} C_VEL
LIN {X 0,Y 378.115,Z 162.409,A -85,B 0,C 180,E1 -12510.998,E2 -12510.998} C_VEL
LIN {X 0,Y 380.197,Z 170.207,A -85,B 0,C 180,E1 -12511.29,E2 -12511.29} C_VEL
LIN {X 0,Y 383.491,Z 186.507,A -85,B 0,C 180,E1 -12511.793,E2 -12511.793} C_VEL
LIN {X 0,Y 382.103,Z 269.618,A -85,B 0,C 180,E1 -12513.394,E2 -12513.394} C_VEL
LIN {X 0,Y 381.606,Z 282.224,A -85,B 0,C 180,E1 -12513.828,E2 -12513.828} C_VEL
LIN {X 0,Y 381.015,Z 295.146,A -85,B 0,C 180,E1 -12514.496,E2 -12514.496} C_VEL
LIN {X 0,Y 380.281,Z 306.669,A -85,B 0,C 180,E1 -12515.302,E2 -12515.302} C_VEL
LIN {X 0,Y 379.39,Z 318.488,A -85,B 0,C 180,E1 -12516.381,E2 -12516.381} C_VEL
LIN {X 0,Y 378.458,Z 329.122,A -85,B 0,C 180,E1 -12517.603,E2 -12517.603} C_VEL
LIN {X 0,Y 377.638,Z 337.699,A -85,B 0,C 180,E1 -12518.815,E2 -12518.815} C_VEL
LIN {X 0,Y 376.834,Z 345.794,A -85,B 0,C 180,E1 -12520.205,E2 -12520.205} C_VEL
LIN {X 0,Y 376.071,Z 353.566,A -85,B 0,C 180,E1 -12521.863,E2 -12521.863} C_VEL
LIN {X 0,Y 375.449,Z 360.14,A -85,B 0,C 180,E1 -12523.63,E2 -12523.63} C_VEL
LIN {X 0,Y 375.07,Z 364.724,A -85,B 0,C 180,E1 -12525.208,E2 -12525.208} C_VEL
LIN {X 0,Y 374.83,Z 367.486,A -85,B 0,C 180,E1 -12526.399,E2 -12526.399} C_VEL
LIN {X 0,Y 374.006,Z 369.163,A -85,B 0,C 180,E1 -12527.259,E2 -12527.259} C_VEL
LIN {X 0,Y 370.947,Z 371.392,A -85,B 0,C 180,E1 -12528.67,E2 -12528.67} C_VEL
LIN {X 0,Y 368.43,Z 372.634,A -85,B 0,C 180,E1 -12529.825,E2 -12529.825} C_VEL
LIN {X 0,Y 367.352,Z 373.261,A -85,B 0,C 180,E1 -12530.728,E2 -12530.728} C_VEL
LIN {X 0,Y 367.263,Z 373.39,A -85,B 0,C 180,E1 -12531.035,E2 -12531.035} C_VEL
LIN {X 0,Y 367.326,Z 373.465,A -85,B 0,C 180,E1 -12533.313,E2 -12533.313} C_VEL
LIN {X 0,Y 367.388,Z 372.525,A -85,B 0,C 180,E1 -12534.888,E2 -12534.888} C_VEL
LIN {X 0,Y 367.538,Z 371.21,A -85,B 0,C 180,E1 -12536.091,E2 -12536.091} C_VEL
LIN {X 0,Y 367.852,Z 368.303,A -85,B 0,C 180,E1 -12537.91,E2 -12537.91} C_VEL
LIN {X 0,Y 368.247,Z 364.119,A -85,B 0,C 180,E1 -12539.75,E2 -12539.75} C_VEL
LIN {X 0,Y 368.865,Z 358.497,A -85,B 0,C 180,E1 -12541.598,E2 -12541.598} C_VEL
LIN {X 0,Y 369.716,Z 351.122,A -85,B 0,C 180,E1 -12543.454,E2 -12543.454} C_VEL
LIN {X 0,Y 370.72,Z 342.488,A -85,B 0,C 180,E1 -12545.171,E2 -12545.171} C_VEL
LIN {X 0,Y 371.783,Z 332.66,A -85,B 0,C 180,E1 -12546.714,E2 -12546.714} C_VEL
LIN {X 0,Y 372.945,Z 321.934,A -85,B 0,C 180,E1 -12548.059,E2 -12548.059} C_VEL
LIN {X 0,Y 373.956,Z 310.455,A -85,B 0,C 180,E1 -12549.193,E2 -12549.193} C_VEL
LIN {X 0,Y 374.977,Z 298.153,A -85,B 0,C 180,E1 -12550.13,E2 -12550.13} C_VEL
LIN {X 0,Y 375.642,Z 285.311,A -85,B 0,C 180,E1 -12550.858,E2 -12550.858} C_VEL
LIN {X 0,Y 376.147,Z 271.758,A -85,B 0,C 180,E1 -12551.37,E2 -12551.37} C_VEL
LIN {X 0,Y 376.875,Z 237.306,A -85,B 0,C 180,E1 -12552.076,E2 -12552.076} C_VEL
LIN {X 0,Y 377.683,Z 186.983,A -85,B 0,C 180,E1 -12553.066,E2 -12553.066} C_VEL
LIN {X 0,Y 374.447,Z 171.98,A -85,B 0,C 180,E1 -12553.588,E2 -12553.588} C_VEL
LIN {X 0,Y 371.174,Z 163.144,A -85,B 0,C 180,E1 -12554.013,E2 -12554.013} C_VEL
LIN {X 0,Y 368.992,Z 152.521,A -85,B 0,C 180,E1 -12556.949,E2 -12556.949} C_VEL
LIN {X 0,Y 368.949,Z 152.535,A -85,B 0,C 180,E1 -12559.636,E2 -12559.636} C_VEL
LIN {X 0,Y 368.9,Z 152.538,A -85,B 0,C 180,E1 -12563.145,E2 -12563.145} C_VEL
LIN {X 0,Y 368.893,Z 152.533,A -85,B 0,C 180,E1 -12566.463,E2 -12566.463} C_VEL
LIN {X 0,Y 368.926,Z 152.53,A -85,B 0,C 180,E1 -12569.047,E2 -12569.047} C_VEL
LIN {X 0,Y 368.978,Z 152.527,A -85,B 0,C 180,E1 -12571.565,E2 -12571.565} C_VEL
LIN {X 0,Y 368.998,Z 152.523,A -85,B 0,C 180,E1 -12574.021,E2 -12574.021} C_VEL
LIN {X 0,Y 368.932,Z 152.531,A -85,B 0,C 180,E1 -12577.606,E2 -12577.606} C_VEL
LIN {X 0,Y 368.953,Z 152.529,A -85,B 0,C 180,E1 -12581.107,E2 -12581.107} C_VEL
LIN {X 0,Y 368.997,Z 152.521,A -85,B 0,C 180,E1 -12584.536,E2 -12584.536} C_VEL
LIN {X 0,Y 369.005,Z 152.516,A -85,B 0,C 180,E1 -12587.908,E2 -12587.908} C_VEL
LIN {X 0,Y 369.091,Z 152.501,A -85,B 0,C 180,E1 -12591.239,E2 -12591.239} C_VEL
LIN {X 0,Y 369.132,Z 152.501,A -85,B 0,C 180,E1 -12594.538,E2 -12594.538} C_VEL
LIN {X 0,Y 369.315,Z 152.476,A -85,B 0,C 180,E1 -12597.82,E2 -12597.82} C_VEL
LIN {X 0,Y 369.432,Z 152.46,A -85,B 0,C 180,E1 -12600.001,E2 -12600.001} C_VEL
LIN {X 0,Y 369.304,Z 152.476,A -85,B 0,C 180,E1 -12602.182,E2 -12602.182} C_VEL
LIN {X 0,Y 369.162,Z 152.492,A -85,B 0,C 180,E1 -12606.56,E2 -12606.56} C_VEL
LIN {X 0,Y 369.065,Z 152.508,A -85,B 0,C 180,E1 -12609.869,E2 -12609.869} C_VEL
LIN {X 0,Y 369.04,Z 152.517,A -85,B 0,C 180,E1 -12613.773,E2 -12613.773} C_VEL
LIN {X 0,Y 368.98,Z 152.519,A -85,B 0,C 180,E1 -12617.757,E2 -12617.757} C_VEL
LIN {X 0,Y 368.911,Z 152.525,A -85,B 0,C 180,E1 -12621.222,E2 -12621.222} C_VEL
LIN {X 0,Y 368.91,Z 152.533,A -85,B 0,C 180,E1 -12623.874,E2 -12623.874} C_VEL
LIN {X 0,Y 368.859,Z 152.533,A -85,B 0,C 180,E1 -12627.213,E2 -12627.213} C_VEL
LIN {X 0,Y 368.893,Z 152.529,A -85,B 0,C 180,E1 -12629.693,E2 -12629.693} C_VEL
LIN {X 0,Y 368.897,Z 152.535,A -85,B 0,C 180,E1 -12633.043,E2 -12633.043} C_VEL
LIN {X 0,Y 368.912,Z 152.53,A -85,B 0,C 180,E1 -12636.198,E2 -12636.198} C_VEL
LIN {X 0,Y 368.874,Z 152.535,A -85,B 0,C 180,E1 -12638.958,E2 -12638.958} C_VEL
LIN {X 0,Y 368.86,Z 152.539,A -85,B 0,C 180,E1 -12642.006,E2 -12642.006} C_VEL
LIN {X 0,Y 368.876,Z 152.543,A -85,B 0,C 180,E1 -12645.175,E2 -12645.175} C_VEL
LIN {X 0,Y 368.863,Z 152.542,A -85,B 0,C 180,E1 -12648.175,E2 -12648.175} C_VEL
LIN {X 0,Y 368.879,Z 152.537,A -85,B 0,C 180,E1 -12651.367,E2 -12651.367} C_VEL
LIN {X 0,Y 368.938,Z 152.528,A -85,B 0,C 180,E1 -12655.147,E2 -12655.147} C_VEL
LIN {X 0,Y 368.899,Z 152.535,A -85,B 0,C 180,E1 -12659.044,E2 -12659.044} C_VEL
LIN {X 0,Y 368.956,Z 152.698,A -85,B 0,C 180,E1 -12659.92,E2 -12659.92} C_VEL
LIN {X 0,Y 371.424,Z 163.967,A -85,B 0,C 180,E1 -12662.79,E2 -12662.79} C_VEL
LIN {X 0,Y 372.889,Z 172.145,A -85,B 0,C 180,E1 -12664.781,E2 -12664.781} C_VEL
LIN {X 0,Y 371.861,Z 184.459,A -85,B 0,C 180,E1 -12667.498,E2 -12667.498} C_VEL
LIN {X 0,Y 371.563,Z 187.053,A -85,B 0,C 180,E1 -12668.061,E2 -12668.061} C_VEL
LIN {X 0,Y 375.85,Z 211.378,A -85,B 0,C 180,E1 -12668.853,E2 -12668.853} C_VEL
LIN {X 0,Y 377.209,Z 221.469,A -85,B 0,C 180,E1 -12669.146,E2 -12669.146} C_VEL
LIN {X 0,Y 376.023,Z 295.716,A -85,B 0,C 180,E1 -12670.625,E2 -12670.625} C_VEL
LIN {X 0,Y 375.276,Z 308.907,A -85,B 0,C 180,E1 -12671.082,E2 -12671.082} C_VEL
LIN {X 0,Y 374.351,Z 321.621,A -85,B 0,C 180,E1 -12671.743,E2 -12671.743} C_VEL
LIN {X 0,Y 373.333,Z 333.75,A -85,B 0,C 180,E1 -12672.612,E2 -12672.612} C_VEL
LIN {X 0,Y 372.186,Z 345.298,A -85,B 0,C 180,E1 -12673.687,E2 -12673.687} C_VEL
LIN {X 0,Y 371.236,Z 354.93,A -85,B 0,C 180,E1 -12674.809,E2 -12674.809} C_VEL
LIN {X 0,Y 370.209,Z 365.106,A -85,B 0,C 180,E1 -12676.273,E2 -12676.273} C_VEL
LIN {X 0,Y 369.169,Z 374.194,A -85,B 0,C 180,E1 -12677.912,E2 -12677.912} C_VEL
LIN {X 0,Y 368.445,Z 381.534,A -85,B 0,C 180,E1 -12679.56,E2 -12679.56} C_VEL
LIN {X 0,Y 367.963,Z 387.426,A -85,B 0,C 180,E1 -12681.211,E2 -12681.211} C_VEL
LIN {X 0,Y 367.6,Z 392.073,A -85,B 0,C 180,E1 -12682.862,E2 -12682.862} C_VEL
LIN {X 0,Y 367.447,Z 395.618,A -85,B 0,C 180,E1 -12684.512,E2 -12684.512} C_VEL
LIN {X 0,Y 367.452,Z 397.411,A -85,B 0,C 180,E1 -12685.612,E2 -12685.612} C_VEL
LIN {X 0,Y 367.398,Z 399.744,A -85,B 0,C 180,E1 -12687.808,E2 -12687.808} C_VEL
LIN {X 0,Y 367.47,Z 400.322,A -85,B 0,C 180,E1 -12688.904,E2 -12688.904} C_VEL
LIN {X 0,Y 367.509,Z 400.464,A -85,B 0,C 180,E1 -12690,E2 -12690} C_VEL
LIN {X 0,Y 367.487,Z 400.201,A -85,B 0,C 180,E1 -12691.096,E2 -12691.096} C_VEL
LIN {X 0,Y 367.384,Z 398.498,A -85,B 0,C 180,E1 -12693.29,E2 -12693.29} C_VEL
LIN {X 0,Y 367.452,Z 396.999,A -85,B 0,C 180,E1 -12694.388,E2 -12694.388} C_VEL
LIN {X 0,Y 367.466,Z 394.054,A -85,B 0,C 180,E1 -12695.991,E2 -12695.991} C_VEL
LIN {X 0,Y 367.697,Z 389.826,A -85,B 0,C 180,E1 -12697.689,E2 -12697.689} C_VEL
LIN {X 0,Y 368.123,Z 383.507,A -85,B 0,C 180,E1 -12699.617,E2 -12699.617} C_VEL
LIN {X 0,Y 368.679,Z 376.622,A -85,B 0,C 180,E1 -12701.268,E2 -12701.268} C_VEL
LIN {X 0,Y 369.588,Z 368.03,A -85,B 0,C 180,E1 -12702.911,E2 -12702.911} C_VEL
LIN {X 0,Y 370.453,Z 359.193,A -85,B 0,C 180,E1 -12704.278,E2 -12704.278} C_VEL
LIN {X 0,Y 371.39,Z 348.31,A -85,B 0,C 180,E1 -12705.644,E2 -12705.644} C_VEL
LIN {X 0,Y 372.399,Z 337.383,A -85,B 0,C 180,E1 -12706.727,E2 -12706.727} C_VEL
LIN {X 0,Y 373.41,Z 325.129,A -85,B 0,C 180,E1 -12707.668,E2 -12707.668} C_VEL
LIN {X 0,Y 374.339,Z 312.282,A -85,B 0,C 180,E1 -12708.4,E2 -12708.4} C_VEL
LIN {X 0,Y 375.005,Z 299.366,A -85,B 0,C 180,E1 -12708.897,E2 -12708.897} C_VEL
LIN {X 0,Y 375.41,Z 281.258,A -85,B 0,C 180,E1 -12709.302,E2 -12709.302} C_VEL
LIN {X 0,Y 376.242,Z 220.331,A -85,B 0,C 180,E1 -12710.489,E2 -12710.489} C_VEL
LIN {X 0,Y 371.17,Z 187.784,A -85,B 0,C 180,E1 -12711.444,E2 -12711.444} C_VEL
LIN {X 0,Y 372.481,Z 173.736,A -85,B 0,C 180,E1 -12714.526,E2 -12714.526} C_VEL
LIN {X 0,Y 372.486,Z 170.127,A -85,B 0,C 180,E1 -12715.345,E2 -12715.345} C_VEL
LIN {X 0,Y 370.056,Z 157.804,A -85,B 0,C 180,E1 -12718.346,E2 -12718.346} C_VEL
LIN {X 0,Y 368.936,Z 152.532,A -85,B 0,C 180,E1 -12719.689,E2 -12719.689} C_VEL
LIN {X 0,Y 368.9,Z 152.536,A -85,B 0,C 180,E1 -12723.538,E2 -12723.538} C_VEL
LIN {X 0,Y 368.904,Z 152.53,A -85,B 0,C 180,E1 -12726.855,E2 -12726.855} C_VEL
LIN {X 0,Y 368.888,Z 152.531,A -85,B 0,C 180,E1 -12730.374,E2 -12730.374} C_VEL
LIN {X 0,Y 368.884,Z 152.535,A -85,B 0,C 180,E1 -12733.615,E2 -12733.615} C_VEL
LIN {X 0,Y 368.887,Z 152.532,A -85,B 0,C 180,E1 -12736.695,E2 -12736.695} C_VEL
LIN {X 0,Y 368.889,Z 152.533,A -85,B 0,C 180,E1 -12739.648,E2 -12739.648} C_VEL
LIN {X 0,Y 368.902,Z 152.536,A -85,B 0,C 180,E1 -12743.145,E2 -12743.145} C_VEL
LIN {X 0,Y 368.9,Z 152.531,A -85,B 0,C 180,E1 -12746.461,E2 -12746.461} C_VEL
LIN {X 0,Y 368.918,Z 152.533,A -85,B 0,C 180,E1 -12749.045,E2 -12749.045} C_VEL
LIN {X 0,Y 368.917,Z 152.528,A -85,B 0,C 180,E1 -12751.558,E2 -12751.558} C_VEL
LIN {X 0,Y 368.928,Z 152.529,A -85,B 0,C 180,E1 -12755.222,E2 -12755.222} C_VEL
LIN {X 0,Y 368.925,Z 152.53,A -85,B 0,C 180,E1 -12758.98,E2 -12758.98} C_VEL
LIN {X 0,Y 368.958,Z 152.525,A -85,B 0,C 180,E1 -12762.255,E2 -12762.255} C_VEL
LIN {X 0,Y 369.043,Z 152.515,A -85,B 0,C 180,E1 -12766.227,E2 -12766.227} C_VEL
LIN {X 0,Y 369.066,Z 152.512,A -85,B 0,C 180,E1 -12770.131,E2 -12770.131} C_VEL
LIN {X 0,Y 369.163,Z 152.497,A -85,B 0,C 180,E1 -12773.44,E2 -12773.44} C_VEL
LIN {X 0,Y 369.306,Z 152.481,A -85,B 0,C 180,E1 -12777.818,E2 -12777.818} C_VEL
LIN {X 0,Y 369.208,Z 152.491,A -85,B 0,C 180,E1 -12781.09,E2 -12781.09} C_VEL
LIN {X 0,Y 369.304,Z 152.486,A -85,B 0,C 180,E1 -12782.18,E2 -12782.18} C_VEL
LIN {X 0,Y 369.158,Z 152.499,A -85,B 0,C 180,E1 -12786.558,E2 -12786.558} C_VEL
LIN {X 0,Y 369.06,Z 152.515,A -85,B 0,C 180,E1 -12789.867,E2 -12789.867} C_VEL
LIN {X 0,Y 369.039,Z 152.517,A -85,B 0,C 180,E1 -12793.771,E2 -12793.771} C_VEL
LIN {X 0,Y 368.955,Z 152.529,A -85,B 0,C 180,E1 -12797.744,E2 -12797.744} C_VEL
LIN {X 0,Y 368.909,Z 152.53,A -85,B 0,C 180,E1 -12801.22,E2 -12801.22} C_VEL
LIN {X 0,Y 368.908,Z 152.533,A -85,B 0,C 180,E1 -12803.873,E2 -12803.873} C_VEL
LIN {X 0,Y 368.857,Z 152.538,A -85,B 0,C 180,E1 -12807.211,E2 -12807.211} C_VEL
LIN {X 0,Y 368.892,Z 152.535,A -85,B 0,C 180,E1 -12809.691,E2 -12809.691} C_VEL
LIN {X 0,Y 368.895,Z 152.533,A -85,B 0,C 180,E1 -12813.042,E2 -12813.042} C_VEL
LIN {X 0,Y 368.914,Z 152.528,A -85,B 0,C 180,E1 -12816.196,E2 -12816.196} C_VEL
LIN {X 0,Y 368.871,Z 152.536,A -85,B 0,C 180,E1 -12818.956,E2 -12818.956} C_VEL
LIN {X 0,Y 368.861,Z 152.535,A -85,B 0,C 180,E1 -12822.005,E2 -12822.005} C_VEL
LIN {X 0,Y 368.871,Z 152.54,A -85,B 0,C 180,E1 -12825.174,E2 -12825.174} C_VEL
LIN {X 0,Y 368.865,Z 152.534,A -85,B 0,C 180,E1 -12828.174,E2 -12828.174} C_VEL
LIN {X 0,Y 368.873,Z 152.536,A -85,B 0,C 180,E1 -12831.365,E2 -12831.365} C_VEL
LIN {X 0,Y 368.926,Z 152.53,A -85,B 0,C 180,E1 -12835.145,E2 -12835.145} C_VEL
LIN {X 0,Y 368.907,Z 152.533,A -85,B 0,C 180,E1 -12839.044,E2 -12839.044} C_VEL
LIN {X 0,Y 368.901,Z 152.53,A -85,B 0,C 180,E1 -12841.557,E2 -12841.557} C_VEL
LIN {X 0,Y 368.88,Z 152.533,A -85,B 0,C 180,E1 -12845.219,E2 -12845.219} C_VEL
LIN {X 0,Y 368.89,Z 152.531,A -85,B 0,C 180,E1 -12847.602,E2 -12847.602} C_VEL
LIN {X 0,Y 368.907,Z 152.53,A -85,B 0,C 180,E1 -12851.103,E2 -12851.103} C_VEL
LIN {X 0,Y 368.932,Z 152.531,A -85,B 0,C 180,E1 -12854.532,E2 -12854.532} C_VEL
LIN {X 0,Y 369.05,Z 152.513,A -85,B 0,C 180,E1 -12856.79,E2 -12856.79} C_VEL
LIN {X 0,Y 369.05,Z 152.516,A -85,B 0,C 180,E1 -12860.131,E2 -12860.131} C_VEL
LIN {X 0,Y 369.15,Z 152.499,A -85,B 0,C 180,E1 -12863.441,E2 -12863.441} C_VEL
LIN {X 0,Y 369.296,Z 152.593,A -85,B 0,C 180,E1 -12867.887,E2 -12867.887} C_VEL
LIN {X 0,Y 371.016,Z 162.71,A -85,B 0,C 180,E1 -12870.619,E2 -12870.619} C_VEL
LIN {X 0,Y 373.314,Z 170.436,A -85,B 0,C 180,E1 -12870.913,E2 -12870.913} C_VEL
LIN {X 0,Y 376.796,Z 188.026,A -85,B 0,C 180,E1 -12871.467,E2 -12871.467} C_VEL
LIN {X 0,Y 375.286,Z 270.498,A -85,B 0,C 180,E1 -12873.087,E2 -12873.087} C_VEL
LIN {X 0,Y 374.77,Z 283.605,A -85,B 0,C 180,E1 -12873.561,E2 -12873.561} C_VEL
LIN {X 0,Y 374.174,Z 296.218,A -85,B 0,C 180,E1 -12874.241,E2 -12874.241} C_VEL
LIN {X 0,Y 373.349,Z 308.53,A -85,B 0,C 180,E1 -12875.149,E2 -12875.149} C_VEL
LIN {X 0,Y 372.444,Z 319.867,A -85,B 0,C 180,E1 -12876.229,E2 -12876.229} C_VEL
LIN {X 0,Y 371.481,Z 330.295,A -85,B 0,C 180,E1 -12877.473,E2 -12877.473} C_VEL
LIN {X 0,Y 370.488,Z 339.954,A -85,B 0,C 180,E1 -12878.916,E2 -12878.916} C_VEL
LIN {X 0,Y 369.638,Z 348.05,A -85,B 0,C 180,E1 -12880.406,E2 -12880.406} C_VEL
LIN {X 0,Y 368.933,Z 355.464,A -85,B 0,C 180,E1 -12882.096,E2 -12882.096} C_VEL
LIN {X 0,Y 368.304,Z 361.399,A -85,B 0,C 180,E1 -12883.81,E2 -12883.81} C_VEL
LIN {X 0,Y 367.928,Z 365.979,A -85,B 0,C 180,E1 -12885.511,E2 -12885.511} C_VEL
LIN {X 0,Y 367.627,Z 369.222,A -85,B 0,C 180,E1 -12887.091,E2 -12887.091} C_VEL
LIN {X 0,Y 367.375,Z 371.878,A -85,B 0,C 180,E1 -12888.978,E2 -12888.978} C_VEL
LIN {X 0,Y 367.263,Z 373.39,A -85,B 0,C 180,E1 -12891.035,E2 -12891.035} C_VEL
LIN {X 0,Y 366.586,Z 373.69,A -85,B 0,C 180,E1 -12891.951,E2 -12891.951} C_VEL
LIN {X 0,Y 363.744,Z 373.594,A -85,B 0,C 180,E1 -12893.442,E2 -12893.442} C_VEL
LIN {X 0,Y 361.398,Z 372.973,A -85,B 0,C 180,E1 -12894.645,E2 -12894.645} C_VEL
LIN {X 0,Y 360.464,Z 372.19,A -85,B 0,C 180,E1 -12895.569,E2 -12895.569} C_VEL
LIN {X 0,Y 360.427,Z 371.817,A -85,B 0,C 180,E1 -12895.879,E2 -12895.879} C_VEL
LIN {X 0,Y 360.757,Z 368.888,A -85,B 0,C 180,E1 -12897.875,E2 -12897.875} C_VEL
LIN {X 0,Y 361.161,Z 364.817,A -85,B 0,C 180,E1 -12899.75,E2 -12899.75} C_VEL
LIN {X 0,Y 361.808,Z 359.336,A -85,B 0,C 180,E1 -12901.632,E2 -12901.632} C_VEL
LIN {X 0,Y 362.511,Z 353.396,A -85,B 0,C 180,E1 -12903.232,E2 -12903.232} C_VEL
LIN {X 0,Y 363.386,Z 346.265,A -85,B 0,C 180,E1 -12904.788,E2 -12904.788} C_VEL
LIN {X 0,Y 364.514,Z 336.784,A -85,B 0,C 180,E1 -12906.443,E2 -12906.443} C_VEL
LIN {X 0,Y 365.613,Z 327.233,A -85,B 0,C 180,E1 -12907.786,E2 -12907.786} C_VEL
LIN {X 0,Y 366.633,Z 317.6,A -85,B 0,C 180,E1 -12908.887,E2 -12908.887} C_VEL
LIN {X 0,Y 367.684,Z 306.027,A -85,B 0,C 180,E1 -12909.938,E2 -12909.938} C_VEL
LIN {X 0,Y 368.555,Z 294.02,A -85,B 0,C 180,E1 -12910.777,E2 -12910.777} C_VEL
LIN {X 0,Y 369.218,Z 281.681,A -85,B 0,C 180,E1 -12911.411,E2 -12911.411} C_VEL
LIN {X 0,Y 369.663,Z 269.193,A -85,B 0,C 180,E1 -12911.834,E2 -12911.834} C_VEL
LIN {X 0,Y 371.246,Z 188.658,A -85,B 0,C 180,E1 -12913.446,E2 -12913.446} C_VEL
